DATA_BLOCK "Charge_1"	// DB 160
VERSION : 0.1
  STRUCT
   Recipe : INT ;
   batches : DINT ;
   Start : INT ;
   batchtime : DATE_AND_TIME ;
   header : ARRAY  [1 .. 7 ] OF INT ;
   BR : ARRAY  [1 .. 25 ] OF UDT 3;
  END_STRUCT ;	
BEGIN
   Recipe := 99;
   batches := L#8;
   Start := 2;
   BR[1].comp_nr := 4;
   BR[1].rated_val := 1.000000e+01;
   BR[1].real_val := 1.000681e+01;
   BR[3].comp_nr := 5;
   BR[3].rated_val := 5.000000e+00;
   BR[3].real_val := 4.986557e+00;
END_DATA_BLOCK

DATA_BLOCK "Charge_2"	// DB 161
VERSION : 0.1
  STRUCT
   Recipe : INT ;
   batches : DINT ;
   Start : INT ;
   batchtime : DATE_AND_TIME ;
   header : ARRAY  [1 .. 7 ] OF INT ;
   BR : ARRAY  [1 .. 25 ] OF UDT 3;
  END_STRUCT ;	
BEGIN
   Recipe := 199;
   batches := L#5;
   Start := 1;
   BR[1].comp_nr := 2;
   BR[1].rated_val := 2.000000e+00;
   BR[1].real_val := 3.009904e+00;
   BR[2].comp_nr := 3;
   BR[2].rated_val := 2.000000e+00;
   BR[2].real_val := 2.706667e+00;
   BR[3].comp_nr := 4;
   BR[3].rated_val := 2.000000e+00;
   BR[3].real_val := 1.864344e+00;
   BR[4].comp_nr := 6;
   BR[4].rated_val := 2.000000e-01;
   BR[4].real_val := 3.235633e-01;
   BR[5].comp_nr := 7;
   BR[5].rated_val := 2.000000e-01;
   BR[5].real_val := 4.058950e-01;
   BR[6].comp_nr := 8;
   BR[6].rated_val := 2.000000e-01;
   BR[6].real_val := 3.326198e-01;
   BR[7].comp_nr := 9;
   BR[7].rated_val := 2.000000e-01;
   BR[7].real_val := 3.507328e-01;
   BR[8].comp_nr := 10;
   BR[8].rated_val := 2.000000e-01;
   BR[8].real_val := 2.206488e-01;
   BR[9].comp_nr := 11;
   BR[9].rated_val := 2.000000e-01;
   BR[9].real_val := 2.684011e-01;
   BR[11].comp_nr := 5;
   BR[11].rated_val := 5.000000e+00;
   BR[11].real_val := 4.997788e+00;
END_DATA_BLOCK

DATA_BLOCK "Charge_3"	// DB 162
VERSION : 0.1
  STRUCT
   Recipe : INT ;
   batches : DINT ;
   Start : INT ;
   batchtime : DATE_AND_TIME ;
   header : ARRAY  [1 .. 7 ] OF INT ;
   BR : ARRAY  [1 .. 25 ] OF UDT 3;
  END_STRUCT ;	
BEGIN
   Recipe := 199;
   batches := L#6;
   Start := 1;
   BR[1].comp_nr := 2;
   BR[1].rated_val := 2.000000e+00;
   BR[1].real_val := 2.571896e+00;
   BR[2].comp_nr := 3;
   BR[2].rated_val := 2.000000e+00;
   BR[2].real_val := 2.482048e+00;
   BR[3].comp_nr := 4;
   BR[3].rated_val := 2.000000e+00;
   BR[3].real_val := 2.077733e+00;
   BR[4].comp_nr := 6;
   BR[4].rated_val := 2.000000e-01;
   BR[4].real_val := 3.013338e-01;
   BR[5].comp_nr := 7;
   BR[5].rated_val := 2.000000e-01;
   BR[5].real_val := 2.000659e-01;
   BR[6].comp_nr := 8;
   BR[6].rated_val := 2.000000e-01;
   BR[6].real_val := 2.165322e-01;
   BR[7].comp_nr := 9;
   BR[7].rated_val := 2.000000e-01;
   BR[7].real_val := 2.247653e-01;
   BR[8].comp_nr := 10;
   BR[8].rated_val := 2.000000e-01;
   BR[8].real_val := 2.247654e-01;
   BR[9].comp_nr := 11;
   BR[9].rated_val := 2.000000e-01;
   BR[9].real_val := 2.321752e-01;
   BR[11].comp_nr := 5;
   BR[11].rated_val := 5.000000e+00;
   BR[11].real_val := 5.065175e+00;
END_DATA_BLOCK

DATA_BLOCK "Charge_4"	// DB 163
VERSION : 0.1
  STRUCT
   Recipe : INT ;
   batches : DINT ;
   Start : INT ;
   batchtime : DATE_AND_TIME ;
   header : ARRAY  [1 .. 7 ] OF INT ;
   BR : ARRAY  [1 .. 25 ] OF UDT 3;
  END_STRUCT ;	
BEGIN
   Recipe := 199;
   batches := L#7;
   Start := 1;
   BR[1].comp_nr := 2;
   BR[1].rated_val := 2.000000e+00;
   BR[1].real_val := 1.841882e+00;
   BR[2].comp_nr := 3;
   BR[2].rated_val := 2.000000e+00;
   BR[2].real_val := 2.257428e+00;
   BR[3].comp_nr := 4;
   BR[3].rated_val := 2.000000e+00;
   BR[3].real_val := 1.942961e+00;
   BR[4].comp_nr := 6;
   BR[4].rated_val := 2.000000e-01;
   BR[4].real_val := 1.992425e-01;
   BR[5].comp_nr := 7;
   BR[5].rated_val := 2.000000e-01;
   BR[5].real_val := 1.728964e-01;
   BR[6].comp_nr := 8;
   BR[6].rated_val := 2.000000e-01;
   BR[6].real_val := 1.992425e-01;
   BR[7].comp_nr := 9;
   BR[7].rated_val := 2.000000e-01;
   BR[7].real_val := 2.124156e-01;
   BR[8].comp_nr := 10;
   BR[8].rated_val := 2.000000e-01;
   BR[8].real_val := 2.198255e-01;
   BR[9].comp_nr := 11;
   BR[9].rated_val := 2.000000e-01;
   BR[9].real_val := 2.082990e-01;
   BR[11].comp_nr := 5;
   BR[11].rated_val := 5.000000e+00;
   BR[11].real_val := 5.031482e+00;
END_DATA_BLOCK

DATA_BLOCK "Charge_5"	// DB 164
VERSION : 0.1
  STRUCT
   Recipe : INT ;
   batches : DINT ;
   Start : INT ;
   batchtime : DATE_AND_TIME ;
   header : ARRAY  [1 .. 7 ] OF INT ;
   BR : ARRAY  [1 .. 25 ] OF UDT 3;
  END_STRUCT ;	
BEGIN
   Recipe := 199;
   batches := L#1;
   Start := 2;
   BR[1].comp_nr := 2;
   BR[1].rated_val := 2.000000e+00;
   BR[1].real_val := 2.380969e+00;
   BR[2].comp_nr := 4;
   BR[2].rated_val := 2.000000e+00;
   BR[2].real_val := 2.066501e+00;
   BR[3].comp_nr := 6;
   BR[3].rated_val := 2.000000e-01;
   BR[3].real_val := 2.017125e-01;
   BR[4].comp_nr := 7;
   BR[4].rated_val := 2.000000e-01;
   BR[4].real_val := 1.901861e-01;
   BR[5].comp_nr := 8;
   BR[5].rated_val := 2.000000e-01;
   BR[5].real_val := 2.074757e-01;
   BR[6].comp_nr := 9;
   BR[6].rated_val := 2.000000e-01;
   BR[6].real_val := 2.140622e-01;
   BR[7].comp_nr := 10;
   BR[7].rated_val := 2.000000e-01;
   BR[7].real_val := 2.124156e-01;
   BR[8].comp_nr := 11;
   BR[8].rated_val := 2.000000e-01;
   BR[8].real_val := 2.025358e-01;
   BR[10].comp_nr := 5;
   BR[10].rated_val := 5.000000e+00;
   BR[10].real_val := 5.020251e+00;
END_DATA_BLOCK

DATA_BLOCK "Charge_6"	// DB 165
VERSION : 0.1
  STRUCT
   Recipe : INT ;
   batches : DINT ;
   Start : INT ;
   batchtime : DATE_AND_TIME ;
   header : ARRAY  [1 .. 7 ] OF INT ;
   BR : ARRAY  [1 .. 25 ] OF UDT 3;
  END_STRUCT ;	
BEGIN
   Recipe := 199;
   batches := L#2;
   Start := 2;
   BR[1].comp_nr := 2;
   BR[1].rated_val := 2.000000e+00;
   BR[1].real_val := 2.223735e+00;
   BR[2].comp_nr := 4;
   BR[2].rated_val := 2.000000e+00;
   BR[2].real_val := 2.066501e+00;
   BR[3].comp_nr := 6;
   BR[3].rated_val := 2.000000e-01;
   BR[3].real_val := 2.041824e-01;
   BR[4].comp_nr := 7;
   BR[4].rated_val := 2.000000e-01;
   BR[4].real_val := 2.848674e-01;
   BR[5].comp_nr := 8;
   BR[5].rated_val := 2.000000e-01;
   BR[5].real_val := 2.033591e-01;
   BR[6].comp_nr := 9;
   BR[6].rated_val := 2.000000e-01;
   BR[6].real_val := 2.041825e-01;
   BR[7].comp_nr := 10;
   BR[7].rated_val := 2.000000e-01;
   BR[7].real_val := 2.074757e-01;
   BR[8].comp_nr := 11;
   BR[8].rated_val := 2.000000e-01;
   BR[8].real_val := 2.017125e-01;
   BR[10].comp_nr := 5;
   BR[10].rated_val := 5.000000e+00;
   BR[10].real_val := 4.930403e+00;
END_DATA_BLOCK

DATA_BLOCK "Charge_7"	// DB 166
VERSION : 0.1
  STRUCT
   Recipe : INT ;
   batches : DINT ;
   Start : INT ;
   batchtime : DATE_AND_TIME ;
   header : ARRAY  [1 .. 7 ] OF INT ;
   BR : ARRAY  [1 .. 25 ] OF UDT 3;
  END_STRUCT ;	
BEGIN
   Recipe := 199;
   batches := L#3;
   Start := 2;
   BR[1].comp_nr := 2;
   BR[1].rated_val := 2.000000e+00;
   BR[1].real_val := 2.111425e+00;
   BR[2].comp_nr := 4;
   BR[2].rated_val := 2.000000e+00;
   BR[2].real_val := 1.886806e+00;
   BR[3].comp_nr := 6;
   BR[3].rated_val := 2.000000e-01;
   BR[3].real_val := 1.992425e-01;
   BR[4].comp_nr := 7;
   BR[4].rated_val := 2.000000e-01;
   BR[4].real_val := 2.404084e-01;
   BR[5].comp_nr := 8;
   BR[5].rated_val := 2.000000e-01;
   BR[5].real_val := 2.066524e-01;
   BR[6].comp_nr := 9;
   BR[6].rated_val := 2.000000e-01;
   BR[6].real_val := 2.017125e-01;
   BR[7].comp_nr := 10;
   BR[7].rated_val := 2.000000e-01;
   BR[7].real_val := 2.074757e-01;
   BR[8].comp_nr := 11;
   BR[8].rated_val := 2.000000e-01;
   BR[8].real_val := 1.992426e-01;
   BR[10].comp_nr := 5;
   BR[10].rated_val := 5.000000e+00;
   BR[10].real_val := 4.975327e+00;
END_DATA_BLOCK

DATA_BLOCK "Charge_8"	// DB 167
VERSION : 0.1
  STRUCT
   Recipe : INT ;
   batches : DINT ;
   Start : INT ;
   batchtime : DATE_AND_TIME ;
   header : ARRAY  [1 .. 7 ] OF INT ;
   BR : ARRAY  [1 .. 25 ] OF UDT 3;
  END_STRUCT ;	
BEGIN
   Recipe := 2;
   batches := L#11;
   Start := 1;
   BR[1].comp_nr := 3;
   BR[1].rated_val := 2.000000e+01;
   BR[1].real_val := -3.369296e-02;
END_DATA_BLOCK

DATA_BLOCK "Charge_9"	// DB 168
VERSION : 0.1
  STRUCT
   Recipe : INT ;
   batches : DINT ;
   Start : INT ;
   batchtime : DATE_AND_TIME ;
   header : ARRAY  [1 .. 7 ] OF INT ;
   BR : ARRAY  [1 .. 25 ] OF UDT 3;
  END_STRUCT ;	
BEGIN
   Recipe := 2;
   batches := L#12;
   Start := 1;
   BR[1].comp_nr := 6;
   BR[1].rated_val := 1.000000e+00;
END_DATA_BLOCK

DATA_BLOCK "Charge_10"	// DB 169
VERSION : 0.1
  STRUCT
   Recipe : INT ;
   batches : DINT ;
   Start : INT ;
   batchtime : DATE_AND_TIME ;
   header : ARRAY  [1 .. 7 ] OF INT ;
   BR : ARRAY  [1 .. 25 ] OF UDT 3;
  END_STRUCT ;	
BEGIN
   Recipe := 99;
   batches := L#7;
   Start := 2;
   BR[1].comp_nr := 4;
   BR[1].rated_val := 1.000000e+01;
   BR[1].real_val := 1.002927e+01;
   BR[3].comp_nr := 5;
   BR[3].rated_val := 5.000000e+00;
   BR[3].real_val := 4.952865e+00;
END_DATA_BLOCK

DATA_BLOCK "Recipes1-50"	// DB 333
TITLE = Data block for recipes 1-50
//it must be unlinked
//
AUTHOR : Fromm
VERSION : 1.0
  STRUCT
   Rezept : ARRAY  [1 .. 50 ] OF STRUCT
    step : ARRAY  [1 .. 25 ] OF UDT 1;
   END_STRUCT ;
  END_STRUCT ;	
BEGIN
END_DATA_BLOCK

DATA_BLOCK "Recipes51-100"	// DB 334
TITLE = Data block for recipes 51-100
//it must be unlinked
//
VERSION : 0.0
  STRUCT
   Rezept : ARRAY  [51 .. 100 ] OF STRUCT
    step : ARRAY  [1 .. 25 ] OF UDT 1;
   END_STRUCT ;
  END_STRUCT ;	
BEGIN
END_DATA_BLOCK

DATA_BLOCK "Recipes101-150"	// DB 335
TITLE = Data block for recipes 101-150
//it must be unlinked
//
AUTHOR : Fromm
VERSION : 1.0
  STRUCT
   Rezept : ARRAY  [101 .. 150 ] OF STRUCT
    step : ARRAY  [1 .. 25 ] OF UDT 1;
   END_STRUCT ;
  END_STRUCT ;	
BEGIN
END_DATA_BLOCK

DATA_BLOCK "Recipes151-200"	// DB 336
TITLE = Data block for recipes 151-200
//it must be unlinked
//
AUTHOR : Fromm
VERSION : 1.0
  STRUCT
   Rezept : ARRAY  [151 .. 200 ] OF STRUCT
    step : ARRAY  [1 .. 25 ] OF UDT 1;
   END_STRUCT ;
  END_STRUCT ;	
BEGIN
END_DATA_BLOCK

ORGANIZATION_BLOCK OB 1
TITLE = "Main Program Sweep (Cycle)"
VERSION : 0.1
VAR_TEMP
  OB1_EV_CLASS : BYTE ;	//Bits 0-3 = 1 (Coming event), Bits 4-7 = 1 (Event class 1)
  OB1_SCAN_1 : BYTE ;	//1 (Cold restart scan 1 of OB 1), 3 (Scan 2-n of OB 1)
  OB1_PRIORITY : BYTE ;	//Priority of OB Execution
  OB1_OB_NUMBR : BYTE ;	//1 (Organization block 1, OB1)
  OB1_RESERVED_1 : BYTE ;	//Reserved for system
  OB1_RESERVED_2 : BYTE ;	//Reserved for system
  OB1_PREV_CYCLE : INT ;	//Cycle time of previous OB1 scan (milliseconds)
  OB1_MIN_CYCLE : INT ;	//Minimum cycle time of OB1 (milliseconds)
  OB1_MAX_CYCLE : INT ;	//Maximum cycle time of OB1 (milliseconds)
  OB1_DATE_TIME : DATE_AND_TIME ;	//Date and time OB1 started
END_VAR
BEGIN
NETWORK
TITLE =
      A     "permanent_0";
      R     "permanent_0";
      AN    "permanent_1";
      S     "permanent_1";
      A     "Restart_Timer";
      =     "StartupTimer";
      A     "permanent_1";
      FP    M 200.0;
      =     "CPU_Restart";
NETWORK
TITLE =
      CALL  "errors_horn";
      CALL  "start_lamps";
      CALL  "dos_comp_1";
      CALL  "dos_comp_2";
      CALL  "dos_comp_5";
      CALL  "dos_comp_6_SS";
      CALL  "dos_comp_7";
      CALL  "dos_comp_8";
      CALL  "dos_comp_9";
      CALL  "dos_comp_10";
      CALL  "dos_comp_11";
      CALL  "dos_comp_12";
      CALL  "discharge_main_scale";
      CALL  "discharge_sub_scale";
      CALL  "agit_MS";
      CALL  "aigt_level_storage1";
      CALL  "aigt_level_storage2";
      CALL  "filling_vat";
      CALL  "filling_coater";
      CALL  "coater circ";
      CALL  "control_FC";
      CALL  "Hand_OP_FC";
END_ORGANIZATION_BLOCK

ORGANIZATION_BLOCK "I/O_FLT1"	// OB 82
TITLE = "I/O Point Fault"
VERSION : 0.1
VAR_TEMP
  OB82_EV_CLASS : BYTE ;	//16#39, Event class 3, Entering event state, Internal fault event
  OB82_FLT_ID : BYTE ;	//16#XX, Fault identifcation code
  OB82_PRIORITY : BYTE ;	//Priority of OB Execution
  OB82_OB_NUMBR : BYTE ;	//82 (Organization block 82, OB82)
  OB82_RESERVED_1 : BYTE ;	//Reserved for system
  OB82_IO_FLAG : BYTE ;	//Input (01010100), Output (01010101)
  OB82_MDL_ADDR : WORD ;	//Base address of module with fault
  OB82_MDL_DEFECT : BOOL ;	//Module defective
  OB82_INT_FAULT : BOOL ;	//Internal fault
  OB82_EXT_FAULT : BOOL ;	//External fault
  OB82_PNT_INFO : BOOL ;	//Point information
  OB82_EXT_VOLTAGE : BOOL ;	//External voltage low
  OB82_FLD_CONNCTR : BOOL ;	//Field wiring connector missing
  OB82_NO_CONFIG : BOOL ;	//Module has no configuration data
  OB82_CONFIG_ERR : BOOL ;	//Module has configuration error
  OB82_MDL_TYPE : BYTE ;	//Type of module
  OB82_SUB_MDL_ERR : BOOL ;	//Sub-Module is missing or has error
  OB82_COMM_FAULT : BOOL ;	//Communication fault
  OB82_MDL_STOP : BOOL ;	//Module is stopped
  OB82_WTCH_DOG_FLT : BOOL ;	//Watch dog timer stopped module
  OB82_INT_PS_FLT : BOOL ;	//Internal power supply fault
  OB82_PRIM_BATT_FLT : BOOL ;	//Primary battery is in fault
  OB82_BCKUP_BATT_FLT : BOOL ;	//Backup battery is in fault
  OB82_RESERVED_2 : BOOL ;	//Reserved for system
  OB82_RACK_FLT : BOOL ;	//Rack fault, only for bus interface module
  OB82_PROC_FLT : BOOL ;	//Processor fault
  OB82_EPROM_FLT : BOOL ;	//EPROM fault
  OB82_RAM_FLT : BOOL ;	//RAM fault
  OB82_ADU_FLT : BOOL ;	//ADU fault
  OB82_FUSE_FLT : BOOL ;	//Fuse fault
  OB82_HW_INTR_FLT : BOOL ;	//Hardware interupt input in fault
  OB82_RESERVED_3 : BOOL ;	//Reserved for system
  OB82_DATE_TIME : DATE_AND_TIME ;	//Date and time OB82 started
END_VAR
BEGIN
// (block stored without names or comments; labels and parameter names are numbered)
END_ORGANIZATION_BLOCK

ORGANIZATION_BLOCK "RACK_FLT"	// OB 86
TITLE = "Loss Of Rack Fault"
VERSION : 0.1
VAR_TEMP
  OB86_EV_CLASS : BYTE ;	//16#38/39 Event class 3
  OB86_FLT_ID : BYTE ;	//16#C1/C4/C5, Fault identifcation code
  OB86_PRIORITY : BYTE ;	//Priority of OB Execution
  OB86_OB_NUMBR : BYTE ;	//86 (Organization block 86, OB86)
  OB86_RESERVED_1 : BYTE ;	//Reserved for system
  OB86_RESERVED_2 : BYTE ;	//Reserved for system
  OB86_MDL_ADDR : WORD ;	//Base address of IM module in rack with fault
  OB86_RACKS_FLTD : ARRAY  [0 .. 31 ] OF BOOL ;	//Racks in fault
  OB86_DATE_TIME : DATE_AND_TIME ;	//Date and time OB86 started
END_VAR
BEGIN
// (block stored without names or comments; labels and parameter names are numbered)
END_ORGANIZATION_BLOCK

ORGANIZATION_BLOCK "COMPLETE RESTART"	// OB 100
TITLE = "Complete Restart"
VERSION : 0.1
VAR_TEMP
  OB100_EV_CLASS : BYTE ;	//16#13, Event class 1, Entering event state, Event logged in diagnostic buffer
  OB100_STRTUP : BYTE ;	//16#81/82/83/84 Method of startup
  OB100_PRIORITY : BYTE ;	//27 (Priority of 1 is lowest)
  OB100_OB_NUMBR : BYTE ;	//100 (Organization block 100, OB100)
  OB100_RESERVED_1 : BYTE ;	//Reserved for system
  OB100_RESERVED_2 : BYTE ;	//Reserved for system
  OB100_STOP : WORD ;	//Event that caused CPU to stop (16#4xxx)
  OB100_STRT_INFO : DWORD ;	//Information on how system started
  OB100_DATE_TIME : DATE_AND_TIME ;	//Date and time OB100 started
END_VAR
BEGIN
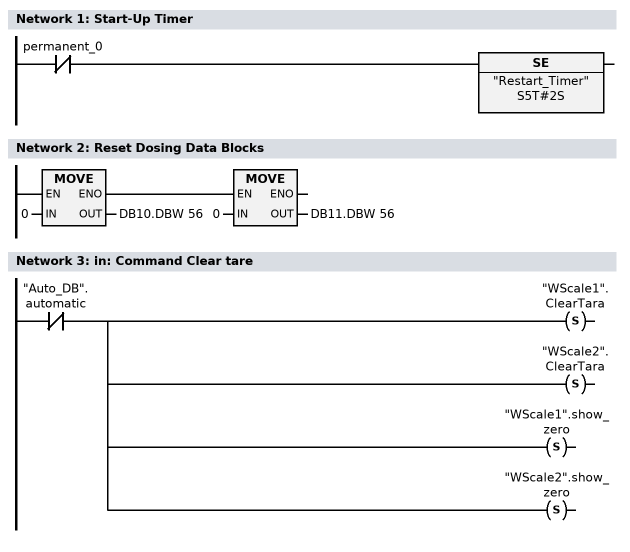
NETWORK
TITLE = Start-Up Timer
      AN    "permanent_0";
      L     S5T#2S;
      SE    "Restart_Timer";
NETWORK
TITLE = Reset Dosing Data Blocks
      A(;
      L     0;
      T     DB10.DBW 56;
      SET;
      SAVE;
      CLR;
      A     BR;
      );
      JNB   _001;
      L     0;
      T     DB11.DBW 56;
_001: NOP   0;
NETWORK
TITLE = in: Command Clear tare
      AN    "Auto_DB".automatic;
      S     "WScale1".ClearTara;
      S     "WScale2".ClearTara;
      S     "WScale1".show_zero;
      S     "WScale2".show_zero;
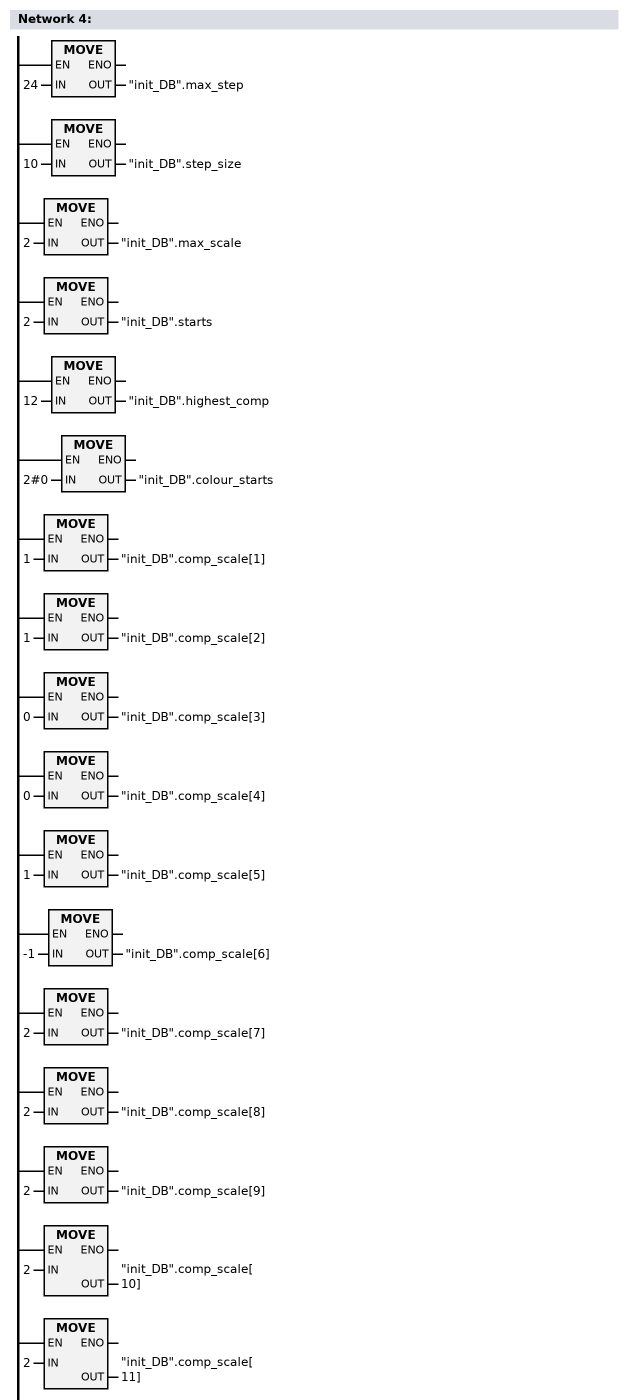
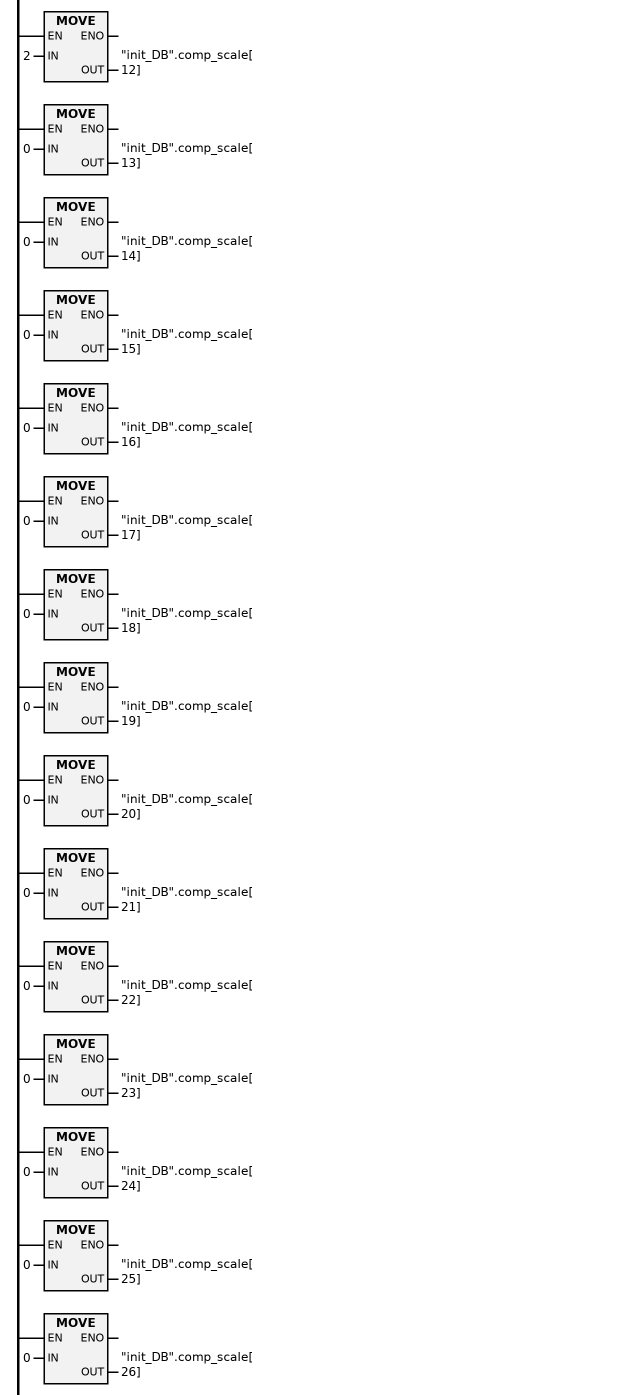
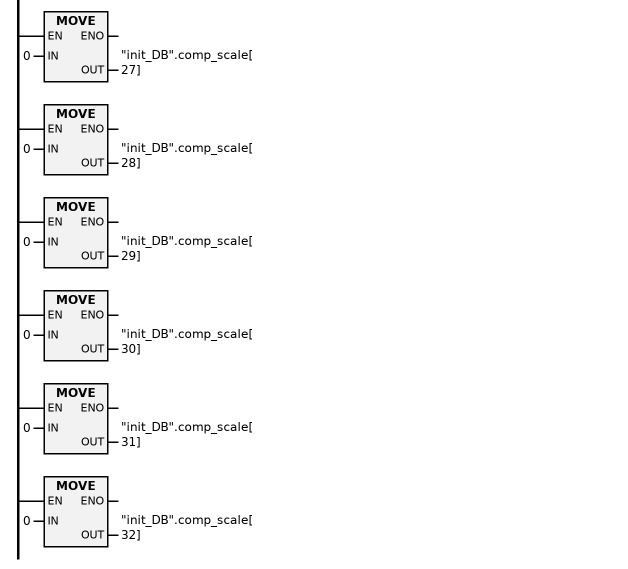
NETWORK
TITLE =
      L     24;
      T     "init_DB".max_step;
      L     10;
      T     "init_DB".step_size;
      L     2;
      T     "init_DB".max_scale;
      L     2;
      T     "init_DB".starts;
      L     12;
      T     "init_DB".highest_comp;
      L     2#0;
      T     "init_DB".colour_starts;
// 1: main scale
// 2: sub scale
// 3: color scale
      L     1;
      T     "init_DB".comp_scale[1];
      L     1;
      T     "init_DB".comp_scale[2];
      L     0;
      T     "init_DB".comp_scale[3];
      L     0;
      T     "init_DB".comp_scale[4];
      L     1;
      T     "init_DB".comp_scale[5];
      L     -1;
      T     "init_DB".comp_scale[6];
      L     2;
      T     "init_DB".comp_scale[7];
      L     2;
      T     "init_DB".comp_scale[8];
      L     2;
      T     "init_DB".comp_scale[9];
      L     2;
      T     "init_DB".comp_scale[10];
      L     2;
      T     "init_DB".comp_scale[11];
      L     2;
      T     "init_DB".comp_scale[12];
      L     0;
      T     "init_DB".comp_scale[13];
      L     0;
      T     "init_DB".comp_scale[14];
      L     0;
      T     "init_DB".comp_scale[15];
      L     0;
      T     "init_DB".comp_scale[16];
      L     0;
      T     "init_DB".comp_scale[17];
      L     0;
      T     "init_DB".comp_scale[18];
      L     0;
      T     "init_DB".comp_scale[19];
      L     0;
      T     "init_DB".comp_scale[20];
      L     0;
      T     "init_DB".comp_scale[21];
      L     0;
      T     "init_DB".comp_scale[22];
      L     0;
      T     "init_DB".comp_scale[23];
      L     0;
      T     "init_DB".comp_scale[24];
      L     0;
      T     "init_DB".comp_scale[25];
      L     0;
      T     "init_DB".comp_scale[26];
      L     0;
      T     "init_DB".comp_scale[27];
      L     0;
      T     "init_DB".comp_scale[28];
      L     0;
      T     "init_DB".comp_scale[29];
      L     0;
      T     "init_DB".comp_scale[30];
      L     0;
      T     "init_DB".comp_scale[31];
      L     0;
      T     "init_DB".comp_scale[32];
NETWORK
TITLE = init CP Gravimet
      L     160;
      T     "init_DB".CP_DB_MIN;
      L     10;
      T     "init_DB".CP_DB_ANZ;
      L     "HMI_DB".CP_DB_WRITE;
      L     "init_DB".CP_DB_MIN;
      <I;
      JC    err1;
      L     "init_DB".CP_DB_MIN;
      L     "init_DB".CP_DB_ANZ;
      +I;
      L     "HMI_DB".CP_DB_WRITE;
      TAK;
      >=I;
      JC    err1;
      JU    go1;
err1: L     "init_DB".CP_DB_MIN;
      T     "HMI_DB".CP_DB_WRITE;
go1:  NOP   0;
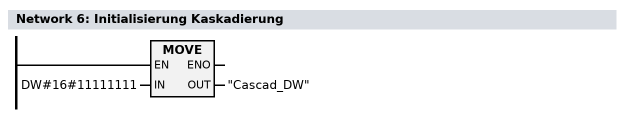
NETWORK
TITLE = Initialisierung Kaskadierung
      L     DW#16#11111111;
      T     "Cascad_DW";
END_ORGANIZATION_BLOCK

ORGANIZATION_BLOCK "PROG_ERR"	// OB 121
TITLE = "Programming Error"
VERSION : 0.1
VAR_TEMP
  OB121_EV_CLASS : BYTE ;	//16#25, Event class 2, Entering event state, Internal fault event
  OB121_SW_FLT : BYTE ;	//16#XX Software programming fault
  OB121_PRIORITY : BYTE ;	//Priority of OB Execution
  OB121_OB_NUMBR : BYTE ;	//121 (Organization block 121, OB121)
  OB121_BLK_TYPE : BYTE ;	//16#88/8A/8B/8C/8E Type of block fault occured in
  OB121_RESERVED_1 : BYTE ;	//Reserved for system
  OB121_FLT_REG : WORD ;	//16#XX Specific register that caused fault
  OB121_BLK_NUM : WORD ;	//Number of block that programming fault occured in
  OB121_PRG_ADDR : WORD ;	//Address in block where programming fault occured
  OB121_DATE_TIME : DATE_AND_TIME ;	//Date and time OB121 started
END_VAR
BEGIN
// (block stored without names or comments; labels and parameter names are numbered)
END_ORGANIZATION_BLOCK

ORGANIZATION_BLOCK "MOD_ERR"	// OB 122
TITLE = "Module Access Error"
VERSION : 0.1
VAR_TEMP
  OB122_EV_CLASS : BYTE ;	//16#29, Event class 2, Entering event state, Internal fault event
  OB122_SW_FLT : BYTE ;	//16#XX Software error code
  OB122_PRIORITY : BYTE ;	//Priority of OB Execution
  OB122_OB_NUMBR : BYTE ;	//122 (Organization block 122, OB122)
  OB122_BLK_TYPE : BYTE ;	//16#88/8C/8E Type of block fault occured in
  OB122_MEM_AREA : BYTE ;	//Memory area where access error occured
  OB122_MEM_ADDR : WORD ;	//Memory address where access error occured
  OB122_BLK_NUM : WORD ;	//Block number in which error occured
  OB122_PRG_ADDR : WORD ;	//Program address where error occured
  OB122_DATE_TIME : DATE_AND_TIME ;	//Date and time OB1 started
END_VAR
BEGIN
// (block stored without names or comments; labels and parameter names are numbered)
END_ORGANIZATION_BLOCK

FUNCTION_BLOCK FB 2
//know_how_protect
//
VERSION : 0.1
VAR_INPUT
  scale_nr : INT ;
  Work_DB : INT ;
  Weigh_DB : INT ;
  mix_timer : TIMER ;
END_VAR
VAR_IN_OUT
  step_scale1 : INT ;
  step_scale2 : INT ;
  step_scale3 : INT ;
  step_scale4 : INT ;
  Dosi_Bits : DINT ;
END_VAR
VAR
  DB_ptr : INT ;
  rated_val : REAL ;
  dosi_val_fine : REAL ;
  dosi_val_coarse : REAL ;
  enable : BOOL ;
  inc_step : BOOL ;
  dosing : BOOL ;
  dosi_coarse : BOOL ;
  dosi_fine : BOOL ;
  cancel : BOOL ;
  discharge : BOOL ;	//out: discharge scale
  wait_still : BOOL ;
  dosi_err : BOOL ;
  dosi_time_err : BOOL ;
  quit_wait : BOOL ;
  redosi : BOOL ;
  mix_time : BOOL ;
  stop : BOOL ;
  clean_out : BOOL ;
  ScaleDosi_Bit : DINT ;
  OwnStep : INT ;
  Status : INT ;
  Rated_Sum : REAL ;
  comp_nr : INT ;
END_VAR
VAR_TEMP
  comp_ok : BOOL ;
  Standstill : BOOL ;
  empty : BOOL ;
  time_empty : BOOL ;
  DosiControl : BOOL ;
  TareScale : BOOL ;
  StepTime : BOOL ;
  ClearTara : BOOL ;
  Temp : INT ;
  NetWeight : REAL ;
  StepPtr : DINT ;
  ScalePtr1 : DINT ;
  scalePtr2 : DINT ;
  scalePtr3 : DINT ;
  scalePtr4 : DINT ;
  t_comp_nr : INT ;
  t_scale : INT ;
  t_spuel : BOOL ;
  start_nr : BYTE ;
END_VAR
BEGIN
NETWORK
TITLE = Read Weighing datas
      L     0;
      T     LB 0;
      AN    #enable;
      BEC;
      L     #Weigh_DB;
      T     #Temp;
      OPN   DB [#Temp];
      L     DBD 88;
      T     #NetWeight;
      A     DBX 58.0;
      =     #Standstill;
      A     DBX 58.3;
      =     #empty;
      A     DBX 58.4;
      =     #time_empty;
      AN    #quit_wait;
      R     #dosi_time_err;
      A     DBX 58.5;
      =     #DosiControl;
      L     0;
      T     #Status;
      A     DBX 58.6;
      =     #StepTime;
      JCN   nost;
      L     10;
      T     #Status;
nost: NOP   0;
      L     #ScaleDosi_Bit;
      L     #Dosi_Bits;
      OD;
      T     #Dosi_Bits;
      A     #cancel;
      R     #quit_wait;
      S     #ClearTara;
NETWORK
TITLE = Jump
      A     #cancel;
      AN    #dosing;
      JC    tend;
      A     #wait_still;
      JC    stil;
      A     #quit_wait;
      JC    end;
      A     #dosi_err;
      JC    t_ok;
      A     #dosing;
      JC    dosi;
      A     #mix_time;
      JC    time;
NETWORK
TITLE = increment own step
      L     #scale_nr;
      L     P#2.0;
      *D;
      L     P#6.0;
      +D;
      T     #StepPtr;
      AN    #inc_step;
      JC    ninc;
      R     #inc_step;
      L     DB1.DBW 0;
      L     #OwnStep;
      ==I;
//      U     #empty
      JC    tend;
// Entleeren, wenn Waage zum Schluß nicht leer (Entleeren vergessen)
// noch nicht ausgereift (Synchronisation fehlt)
//      L     "init_DB".max_step
//      L     #OwnStep
//      ==I   
//      UN    #empty
//      SPB   disc
      INC   1;
      T     DIW [#StepPtr];
      T     #OwnStep;
ninc: NOP   0;
NETWORK
TITLE = calculate pointer
//Vorerst nicht verwendet
      L     #OwnStep;
      DEC   1;
      L     DB1.DBW 2;
      *D;
      SLD   3;
      LAR1;
      L     0;
      L     #step_scale1;
      ==I;
      JC    z1;
      DEC   1;
      L     DB1.DBW 2;
      *D;
      SLD   3;
z1:   T     #ScalePtr1;
      L     0;
      L     #step_scale2;
      ==I;
      JC    z2;
      DEC   1;
      L     DB1.DBW 2;
      *D;
      SLD   3;
z2:   T     #scalePtr2;
      L     0;
      L     #step_scale3;
      ==I;
      JC    z3;
      DEC   1;
      L     DB1.DBW 2;
      *D;
      SLD   3;
z3:   T     #scalePtr3;
      L     0;
      L     #step_scale4;
      ==I;
      JC    z4;
      DEC   1;
      L     DB1.DBW 2;
      *D;
      SLD   3;
z4:   T     #scalePtr4;
NETWORK
TITLE = Sync all other scales
      L     #Work_DB;
      T     #Temp;
      OPN   DB [#Temp];
      L     DBW [AR1,P#2.0];	// comp no.
      T     #t_comp_nr;
      CALL  FC 85 (
           component                := #t_comp_nr,
           scale_nr                 := #t_scale);	//WAAGE FUER KOMPONENTE ABFRAGEN
      A(;
      L     W#16#FF;
      L     #t_scale;
      ==I;	// Spülkomponente
      );
      A(;
      L     #scale_nr;
      L     2;	// Subwaage
      ==I;
      );
      =     #t_spuel;
      A(;
      L     #step_scale1;
      L     #OwnStep;
      <=I;
      );
      A     #t_spuel;
      JC    end;
      L     DBW [AR1,P#0.0];	// Action
      SRW   8;
      L     #scale_nr;
      <>I;
      S     #inc_step;	// nicht für diese Waage
      JC    end;
//      SPA   sync                        // kein Paralleldosieren der waagen
      L     16;
      T     #Status;
      A(;
      L     DBW [AR1,P#0.0];	// Action
      L     W#16#FF;
      AW;
      L     1;	// dosieren
      <=I;
      );
      A(;
      L     #scale_nr;
      L     2;	// nur Subwaage darf parallel
      ==I;
      );
      JC    tar;	// Dosieren ohne Synchronisation (parallel)
      A(;
      L     #step_scale1;
      L     #OwnStep;
      >=I;
      );
      A(;
      L     #step_scale2;
      L     #OwnStep;
      >=I;
      );
      A(;
      L     #step_scale3;
      L     #OwnStep;
      >=I;
      );
      A(;
      L     #step_scale4;
      L     #OwnStep;
      >=I;
      );
      JCN   end;
      NOP   0;
NETWORK
TITLE = step for this scale?
      L     #Work_DB;
      T     #Temp;
      OPN   DB [#Temp];
      L     DBW [AR1,P#0.0];	// Action
      L     W#16#FF;	// nur das untere Byte
      AW;
      T     #Temp;
      L     1;	// dosieren
      <=I;
      JC    tar;
      L     #Temp;	// Action
      L     2;
      ==I;	// mixing?
      JC    mix;
      L     #Temp;	// Action
      L     3;
      ==I;	// discharge?
      JC    disc;
      L     #Temp;	// Action
      L     4;
      ==I;	// discharge cleaning
      S     #clean_out;
      JC    disc;
      S     #inc_step;	// keine der Aktionen
      JU    end;
NETWORK
TITLE = Action: mixing
mix:  L     #OwnStep;
      DEC   1;
      L     DB1.DBW 2;
      *I;
      SLD   3;
      LAR1;
      L     #Work_DB;
      T     #Temp;
      OPN   DB [#Temp];
// Subwaage mit Entleeren
      L     DBW [AR1,P#0.0];	// Action
      L     W#16#FF;
      AW;
      L     0;	// 0 =mit entleeren
      <>I;
      JC    mix2;
      L     W#16#3;
      L     DBW [AR1,P#0.0];
      OW;
      T     DBW [AR1,P#0.0];
      JU    end;
mix2: NOP   0;
// Ende
      L     0;
      L     DBW [AR1,P#4.0];	// mixing time
      ==I;
      S     #inc_step;
      JC    end;
      S     #mix_time;
      JU    end;
time: L     12;
      T     #Status;
      T     LD 34;
      TAK;
      T     LD 38;
      L     #mix_timer;
      T     LW 42;
      L     LD 38;
      L     LD 34;
      AN    T [LW 42];
      BEC;
      SET;
      R     #mix_time;
      S     #inc_step;
      L     0;
      T     #rated_val;
      T     #comp_nr;
      JU    end;
NETWORK
TITLE = Action: discharge scale
disc: L     4;
      T     #Status;
      L     #Rated_Sum;
      T     #rated_val;
      S     #ClearTara;
      A     #empty;
      AN    #time_empty;
      JCN   not;
      L     15;
      T     #Status;
not:  AN    #time_empty;
      =     #discharge;
      JC    end;
      R     #clean_out;
      L     0;
      T     #Rated_Sum;
      JU    mix;
NETWORK
TITLE = tare scale
tar:  L     8;
      T     #Status;
      L     DBW [AR1,P#2.0];	// comp no.
      T     #comp_nr;
      L     DBD [AR1,P#6.0];
      T     #rated_val;
//      CALL  "comp_scale"
//       component:=#comp_nr
//       scale_nr :=#Temp
//      L     #Temp
//      L     #scale_nr
//      <>I   
//      S     #inc_step
//      SPB   end
      L     9;
      T     #Status;
      AN    #Standstill;
      JC    end;
      L     #rated_val;
      L     #Rated_Sum;
      +R;
      T     #Rated_Sum;
      L     #comp_nr;
      L     30;
      +I;
      T     #DB_ptr;
      T     #Temp;
      OPN   DB [#Temp];
      L     1;
      T     #ScaleDosi_Bit;
      L     #comp_nr;
      DEC   1;
      L     #ScaleDosi_Bit;
      SLD;
      T     #ScaleDosi_Bit;
      L     #Dosi_Bits;
      OD;
      T     #Dosi_Bits;
      L     #rated_val;
      L     DBD 16;	// Nachlauf
      -R;
      JP    f_ok;
      L     0.000000e+00;
      T     DBD 16;
      L     #rated_val;
f_ok: T     #dosi_val_fine;
      L     DBD 8;	// grob/fein
      -R;
      JP    c_ok;
//      L     DBD    0
//      T     DBD    8
      L     #dosi_val_fine;
c_ok: T     #dosi_val_coarse;
// DosiTime at CompDatas
      L     DBW 20;
      L     #Weigh_DB;
      T     #Temp;
      TAK;
      OPN   DB [#Temp];
      T     DBW 116;
// End  DosiTime at CompDatas 
      S     #TareScale;
      S     #dosing;
      JU    end;
NETWORK
TITLE = dosing
dosi: A     #cancel;
      JC    t_ok;
      AN    #dosi_fine;
      A     #StepTime;
      JC    end;
      O     #stop;
      O     #DosiControl;
      S     #quit_wait;
      R     #dosi_coarse;
      R     #dosi_fine;
      S     #dosi_time_err;
      JC    end;
      L     #NetWeight;
      L     #dosi_val_fine;
      <R;
      =     #dosi_fine;
      L     #NetWeight;
      L     #dosi_val_coarse;
      <R;
      =     #dosi_coarse;
      L     3;
      A     #dosi_fine;
      AN    #dosi_coarse;
      JC    tran;
      L     2;
tran: T     #Status;
      O     #dosi_coarse;
      O     #dosi_fine;
      JC    end;
NETWORK
TITLE = drip_flow
      A     #StepTime;
      JC    end;
stil: AN    #Standstill;
      =     #wait_still;
      JC    end;
      A     #redosi;
      JC    tol;
      L     #DB_ptr;
      T     #Temp;
      OPN   DB [#Temp];
      L     #NetWeight;
      L     #rated_val;
      -R;
      L     5.000000e-01;
      *R;
      L     DBD 16;
      +R;
      JP    npos;
      L     0.000000e+00;
npos: T     DBD 16;
NETWORK
TITLE = Tolerance
tol:  R     #redosi;
      L     #DB_ptr;
      T     #Temp;
      OPN   DB [#Temp];
      L     #NetWeight;
      L     #rated_val;
      -R;
      JP    tpos;
      S     #redosi;	// evtl nachdos
      ABS;
tpos: L     DBD 12;	// tolerance
      <R;	// Abweichung < Toleranz
      JC    t_ok;
      AN    #redosi;
      S     #dosi_err;
      S     #quit_wait;
      JC    end;
// Nachdosieren
      L     #rated_val;	//neu, Sollwert
      L     DBD 12;	//Toleranz
      -R;
      T     #dosi_val_fine;
      JU    end;
t_ok: R     #dosi_err;
NETWORK
TITLE = dosing end
      R     #dosing;
      CALL  FC 65 (
           start_nr                 := DB21.DBB 6,
           scale_nr                 := #scale_nr,
           step                     := #OwnStep,
           comp                     := #comp_nr,
           rated_val                := #rated_val,
           real_val                 := #NetWeight);
      L     #ScaleDosi_Bit;
      INVD;
      L     #Dosi_Bits;
      AD;
      T     #Dosi_Bits;
      L     0;
      T     #ScaleDosi_Bit;
      A     #cancel;
      JC    tend;
      JU    mix;
NETWORK
TITLE =
tend: L     0;
      T     DIW 34;
      T     #OwnStep;
      T     #Rated_Sum;
      T     #rated_val;
      T     #comp_nr;
NETWORK
TITLE =
end:  A     #mix_time;
      ITB;
      OW    W#16#2000;
      T     LD 34;
      TAK;
      T     LD 38;
      L     #mix_timer;
      T     LW 42;
      L     LD 38;
      L     LD 34;
      SD    T [LW 42];
NETWORK
TITLE = Write Weighing Datas
      L     #Weigh_DB;
      T     #Temp;
      OPN   DB [#Temp];
      A     #TareScale;
      S     DBX 57.0;
      A     #ClearTara;
      S     DBX 57.1;
      A     #dosi_fine;
      =     DBX 57.3;
      A     #discharge;
      =     DBX 57.4;
END_FUNCTION_BLOCK

FUNCTION_BLOCK FB 111
TITLE = Wiegebaustein mit Siwarex CS
//
//Version: 1.0 (Beta-Version)
//Entwicklung: 10.11.2010 Stefan Michel
//
//Bemerkungen: -Baustein für Funktionstests im Haus freigegeben
//             
//
//Änderungen:
//
//
AUTHOR : Michel
VERSION : 1.0
VAR_INPUT
  ADRESSE : INT ;	//Adresse der Siwarex Baugruppe (Hardwarekonfig)
  ABZUGSWAAGE : BOOL ;	//Zuwaage:0;          Abzugswaage:1
  KAS_SIWAREX : BOOL ;	//Kaskadierung Siwarex (wird nur angesprochen, wenn 1 (Zugriffe optimieren)
  CPU_Start_Bit : BOOL ;	//Ein Bit das beim CPU-Start für 1Zyklus den Zustand 1 hat
  ANLAUFTIMER : BOOL ;	//Anlauftimer der CPU
  Quitt : BOOL ;	//Quittiermerker
  StillTimer : TIMER ;	//Timer for Standstill
  EmptyTimer : TIMER ;	//Timer for emptyTime
  DosiControlTimer : TIMER ;	//Timer for dosiControl
  StepTimer : TIMER ;	//Timer for StepTime
END_VAR
VAR_IN_OUT
  SYNCHRON_ERR : BOOL ;	//Synchroner Fehler der SIWAREX
  ASYNCHRON_ERR : BOOL ;	//Asynchroner Fehler der SIWAREX
  SIWA_ERR : BOOL ;	//Siwarex liefert keine neuen Messwerte/oder Kommunikation gestört
  SFB_ERR : BOOL ;	//Fehler bei der SFB-Bearbeitung
  BUSY : BOOL ;	//BIN BESCHÄFTIGT!  Es wird gerade ein SFB abgearbeitet
END_VAR
VAR
  Reserve : ARRAY  [0 .. 1 ] OF //Reserve
  BYTE ;
  AdjustDatas : STRUCT 	//DataRecords 3 and 4
   Zero_set_val_NV : WORD ;	//nicht verwendet
   Meanval_filt_NV : BOOL ;	//nicht verwendet
   EEPROM_NV : BOOL ;	//nicht verwendet
   Chan_active_NV : BOOL ;	//nicht verwendet
   Free1_NV : BOOL ;	//nicht verwendet
   Free2_NV : BOOL ;	//nicht verwendet
   Free3_NV : BOOL ;	//nicht verwendet
   Free4_NV : BOOL ;	//nicht verwendet
   Free5_NV : BOOL ;	//nicht verwendet
   LoadCell1_NV : BOOL ;	//nicht verwendet
   LoadCell2_NV : BOOL ;	//nicht verwendet
   Comma1_NV : BOOL ;	//nicht verwendet
   Comma2_NV : BOOL ;	//nicht verwendet
   Comma3_NV : BOOL ;	//nicht verwendet
   Filter1_NV : BOOL ;	//nicht verwendet
   Filter2_NV : BOOL ;	//nicht verwendet
   Filter3_NV : BOOL ;	//nicht verwendet
   Digit0 : WORD ;	//Adjustment digits dead load
   Digit1 : WORD  := W#16#EA60;	//Adjustment digits Adjustment weight
   AdjustWeight : INT  := 2000;	//Adjustment weight
  END_STRUCT ;
  Reserve_1 : ARRAY  [0 .. 9 ] OF //Reserve
  BYTE ;
  Command : WORD ;	//DataRecords 11 and 12 Command (1 zero point;2 adjustment point; 3 set zero)
  Reserve_2 : ARRAY  [0 .. 7 ] OF //Reserve
  BYTE ;
  ActDatas : STRUCT 	//DataRecords 31 and 32
   Gross : INT ;	//Grossweight für Dosierzeitkontrolle und Stillstandskontrolle
   Status_NV : BYTE ;	//nicht verwendet
   MeasVal_NV : BYTE ;	//nicht verwendet
   Digits : WORD ;
   Asynch_Err_NV : WORD ;	//nicht verwendet
   Synch_Err_NV : WORD ;	//nicht verwendet
  END_STRUCT ;
  ReadAdjust : BOOL ;	//Bit Justagedaten lesen
  Res_1 : BOOL ;
  WriteAdjust : BOOL ;	//Bit Justagedaten schreiben
  Res_2 : BOOL ;
  WriteCommand : BOOL ;	//Write Siwarex command
  Res_3 : BOOL ;
  Res_4 : BOOL ;
  Res_5 : BOOL ;
  TareScale : BOOL ;	//Bit Waage tarieren
  ClearTara : BOOL ;	//Bit lösche Taraspeicher - Zeige Inhalt der Waage
  show_zero : BOOL ;	//zeige absoluten Inhalt der Waage an
  dosing : BOOL ;	//Waage ist in der Dosierung
  discharge : BOOL ;	//Waage ist in der Entleerung
  Res_6 : BOOL ;
  Res_7 : BOOL ;
  Res_8 : BOOL ;
  Standstill : BOOL ;	//Stillstand Waage
  Overload : BOOL ;	//Waage ist überlastet
  no_zero : BOOL ;	//Nullfehler (AbsGewicht > Nullwert)
  empty : BOOL ;	//Erkennung Waage leer --> Leerzeit startet
  time_empty : BOOL ;	//Waage leer und Leerzeit abgelaufen
  DosiControl : BOOL ;	//Dosierzeitfehler
  StepTime : BOOL ;	//Fortschaltezeit läuft
  DosiControl_OldVal : INT ;	//Dosierzeitkontrolle alter Wert
  StandStill_OldVal : INT ;	//Stillstandskontrolle alter Wert
  SiwaWeight : REAL ;	//Absolutwert SIWAREX ohne Nullpunktverschiebung
  spare1 : ARRAY  [1 .. 6 ] OF INT ;
  GrossWeight : REAL ;	//Bruttogewicht
  TareWeight : REAL ;	//Tarierspeicher
  NetWeight : REAL ;	//Nettogewicht
  spare2 : ARRAY  [1 .. 4 ] OF INT ;
  SP : STRUCT
   Range : REAL ;	//Scale range
   zero_val : REAL ;	//Zero value
   empty_val : REAL ;	//empty value
   empty_time : INT ;	//empty time
   step_time : INT ;	//step_time
   DosiControlTime : INT ;	//Time for dosing control
  END_STRUCT ;
  PW_IN : STRUCT 	//Aktuelle Prozesswerte
   KoByte : STRUCT
    NV_1 : BOOL ;
    Befehl_ausgefuehrt : BOOL ;	//Siwarex hat den Befehl empfangen (BI)
    LifeBit : BOOL ;	//LB
    Neustart : BOOL ;	//NEUST
    SyncErr : BOOL ;
    WKGN_Bit0 : BOOL ;
    WKGN_Bit1 : BOOL ;
    WKGN_Bit2 : BOOL ;
   END_STRUCT ;
   Zykluszaehler : BYTE ;	//Zykluszähler
   SyncErrCode : BYTE ;	//synchrone Fehlerinfo (Fehlercode)
   AsyncErr : STRUCT 	//asynchrone Fehlerinfo (Bitweise)
    RAM : BOOL ;	//Neuanlauf wegen RAM-Fehler
    Watchdog : BOOL ;	//Neuanlauf wegen Watchdogfehler
    Programm : BOOL ;	//Neuanlauf wegen Programmfehler
    ueberlaufGewicht : BOOL ;	//Zahlerüberlauf bei Gewichtsberechnung
    Parameter : BOOL ;	//Parameterfehler
    Messbereich : BOOL ;	//AD-Wandler an Messbereichsgrenze
    Drahtbruch : BOOL ;	//Mindestspannung an Sense-Leitung unterschritten
    AD_Wandler : BOOL ;	//AD-Wandlerstörung
   END_STRUCT ;
   Prozesswert : INT ;	//Prozesswert (je nach Auswahl im WKNG)
   Status : STRUCT 	//Status
    Schreibschutz : BOOL ;	//Stellung des Schreibschutzschalters (0=AUS 1=EIN)
    MinWB : BOOL ;	//Min.Wägebereich ist unterschritten
    NV_1 : BOOL ;
    NV_2 : BOOL ;
    NV_3 : BOOL ;
    NV_4 : BOOL ;
    NV_5 : BOOL ;
    BaugruppenErr : BOOL ;	//globale Baugruppenstörung
    GW1 : BOOL ;	//Grenzwert 1 hat angesprochen
    GW2 : BOOL ;	//Grenzwert 2 hat angesprochen
    TaraWaage : BOOL ;	//Waage tariert (Taraspeicher belget)
    TaraExt : BOOL ;	//Taraspeicher mit ext. Vorgabewert belegt
    Max_9E : BOOL ;	//Brutto-Wägebereich mehr als 9 Anzeigeschritte über- oder unterschritten
    _1_4dZero : BOOL ;	//Brutto kleiner +/- 0,25e
    Stillstand : BOOL ;	//Stillstand liegt vor
    Justiert : BOOL ;	//Waage justiert
   END_STRUCT ;
  END_STRUCT ;
  PW_OUT : STRUCT
   KoByte : STRUCT
    NV_B0 : BOOL ;
    BefAusfuehren : BOOL ;	//BIQ
    Quitt_LifeBit : BOOL ;	//LBQ
    Quitt_Neustart : BOOL ;	//Neustart bestätigen (NEUSTQ)
    NV_B4 : BOOL ;
    WKGN_Bit0 : BOOL ;
    WKGN_Bit1 : BOOL ;
    WKGN_Bit2 : BOOL ;
   END_STRUCT ;
   BefNummer : BYTE ;
   Ext_Taravorgabe : INT ;
   NV_Byte4 : BYTE ;	//Nicht verwendet
   NV_Byte5 : BYTE ;	//Nicht verwendet
   NV_Byte6 : BYTE ;	//Nicht verwendet
   NV_Byte7 : BYTE ;	//Nicht verwendet
  END_STRUCT ;
  s_JUST_DAT : STRUCT 	//DR3: Calibration parameters
   w_CALIB_DIGITS0 : WORD ;	//Calibration digits for 0
   w_CALIB_DIGITS1 : WORD  := W#16#EA60;	//Calibration digits for 1
   w_CALIB_DIGITS2 : WORD ;	//Calibration digits for 2
   i_CALIB_WEIGHT1 : INT  := 2000;	//Calibration weight for 1
   i_CALIB_WEIGHT2 : INT ;	//Calibration weight for 2
   b_SIGNAL_RANGE : BYTE  := B#16#2;	//Input range (1=1mV/v, 2=2mV/V, 4=4mV/V)
   b_FILT_TYPE : BYTE ;	//Filter type signal filter (only 0 allowed)
   b_FILT_FREQ : BYTE  := B#16#4;	//Filter low pass frequency
   b_FILT_DEPTH : BYTE  := B#16#F;	//Filter depth of average value filter (0...FF)
   s_SCALE_ID : STRING  [10 ] := 'SIWAREX XX';	//Scale identity
   i_MIN_WR : INT  := 20;	//Minimum for weighing range WR
   i_MAX_WR : INT  := 2000;	//Maximum for weighing range WR
   i_INCREMENT_WR : INT  := 1;	//Digital increment for weighing range
   i_WEIGHT_ST_STILL : INT  := 10;	//Stand still weight
   t_TIME_ST_STILL1 : TIME  := T#1S;	//Stand still time in ms
   b_DEC_POINT : BYTE  := B#16#2;	//Decimal point for remote display
   b_ZERO_NEG_VALUE : BYTE  := B#16#1;	//Zeroing negative range (% of WR)
   b_ZERO_POS_VALUE : BYTE  := B#16#3;	//Zeroing positive range (% of WR)
   b_TARA_MAX : BYTE  := B#16#64;	//Tara range (% of WR)
   i_Reserve : INT ;	//Reserve
   s_LEGAL_TRADE : STRING  [4 ] := '----';	//OIML or no ----
   s_WEGHT_UNIT : STRING  [4 ] := 'kg  ';	//Unit for weight
  END_STRUCT ;
  RDREC_1 : SFB 52;
  WRREC_1 : SFB 53;
  ErrTIMER1_SIWA : SFB 4;	//IEC Timer SFB
  ErrTIMER2_SIWA : SFB 4;	//IEC Timer SFB
  ErrTIMER3_SIWA : SFB 4;	//IEC Timer SFB
  TIMER_Res1 : SFB 4;	//Reserve Timer
  TIMER_Res2 : SFB 4;	//Reserve Timer
  TIMER_Pause : SFB 5;	//Reserve Timer
  TIMER_Res3 : SFB 5;	//Reserve Timer
  CMD_Waage_nullen : BOOL ;	//Bit Waage nullen
  CMD_Res1 : BOOL ;	//Reserve
  CMD_Res2 : BOOL ;	//Bit Allgemeine Parameter schreiben
  CMD_Res3 : BOOL ;	//Bit Befehl an Siwarex ausführen
  CMD_Res4 : BOOL ;	//Bit Befehl an Siwarex ausführen
  CMD_Res5 : BOOL ;	//Bit Befehl an Siwarex ausführen
  CMD_Res6 : BOOL ;	//Bit Befehl an Siwarex ausführen
  CMD_Res7 : BOOL ;	//Bit Befehl an Siwarex ausführen
  REQ_Lese_JustDat : BOOL ;	//SFC ausführen
  REQ_Schreibe_JustDat : BOOL ;	//SFC ausführen
  REQ_Schreibe_Befehl : BOOL ;	//SFC ausführen
  REQ_Res1 : BOOL ;	//Reserve
  REQ_Res2 : BOOL ;	//Reserve
  REQ_Res3 : BOOL ;	//Reserve
  REQ_Res4 : BOOL ;	//SFC ausführen
  REQ_Res5 : BOOL ;	//SFC ausführen
  Urloeschschutz : BOOL ;	//Dieses Bit dient dazu um herauszufiltern ob die CPU urgelöscht wurde
  Simulation : BOOL ;	//Simulationsbetrieb !! Waage ist außer Funktion
  FP_Sim : BOOL ;	//Flankenmerker positive Flanke
  FN_Sim : BOOL ;	//Flankenmerker negative Flanke
  SIM_Wert : WORD ;	//Gewichtswert für die Simulation in [g] (max. 65500g)
  SELECT_PROC_VAL : INT ;
  Nullstellwert : WORD ;	//Nullwert der Waage
  Zykluszaehler_OldVal : INT ;
  RET_VAL_JustDat_lesen : DWORD ;	//Rückgabewert SFC Justagedaten lesen
  RET_VAL_JustDat_schrei : DWORD ;	//Rückgabewert SFC Justagedaten schreiben
  Letzter_SFB_RDErrCode : DWORD ;
  Letzter_SFB_WDErrCode : DWORD ;
  SynchronErrCode : INT ;	//Fehlercode
END_VAR
VAR_TEMP
  T_permanent_0 : BOOL ;	//Dauer 0
  T_permanent_1 : BOOL ;	//Dauer 1
  T_DWORD_ADR : DWORD ;	//Siwarex Baugruppenadresse im DWord-Format
  T_BUSY1 : BOOL ;	//SFB ist beschäftigt
  T_BUSY2 : BOOL ;	//SFB ist beschäftigt
  T_Komma_Fak : REAL ;	//Faktor für die Nachkommastelle
  T_Digit_kg : REAL ;	//Digits pro kg
  T_ToggelMesswert : BOOL ;	//Nach jeden neuen Messwert invertiert die Siwarex dieses Bit
  T_Ptr_KoByte : DINT ;
  T_Ptr_Zykluszaehler : DINT ;
  T_Ptr_SyncErr : DINT ;
  T_Ptr_AsyncErr : DINT ;
  T_Ptr_PW : DINT ;
  T_Ptr_Status : DINT ;
  T_Ptr_PW_OUT : DINT ;
  T_Komma : STRUCT
   Komma1 : BOOL ;
   Komma2 : BOOL ;
   Komma3 : BOOL ;
   NV_1 : BOOL ;
   NV_2 : BOOL ;
   NV_3 : BOOL ;
   NV_4 : BOOL ;
   NV_5 : BOOL ;
  END_STRUCT ;
END_VAR
BEGIN
NETWORK
TITLE = Signal permanent1 und permanent0
      CLR;
      =     #T_permanent_0;
      SET;
      =     #T_permanent_1;
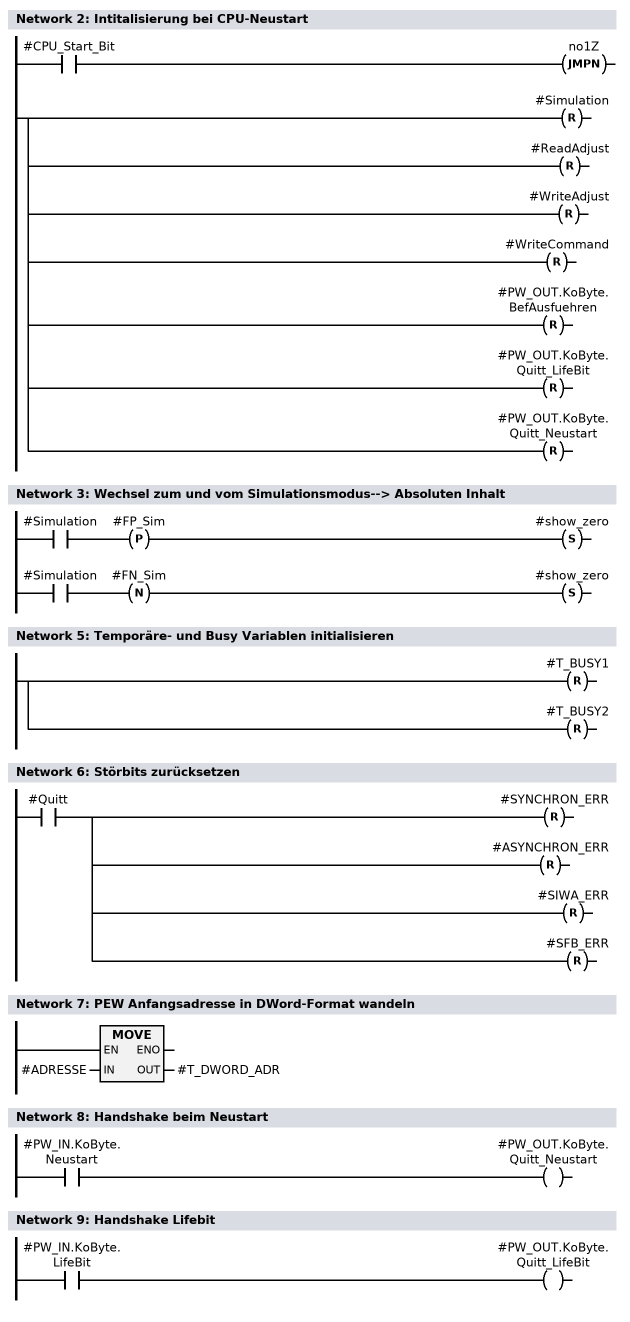
NETWORK
TITLE = Intitalisierung bei CPU-Neustart
//    --------------------------------
      A     #CPU_Start_Bit;
      JCN   no1Z;
      SET;
      R     #Simulation;
      R     #ReadAdjust;
      R     #WriteAdjust;
      R     #WriteCommand;
      R     #PW_OUT.KoByte.BefAusfuehren;
      R     #PW_OUT.KoByte.Quitt_LifeBit;
      R     #PW_OUT.KoByte.Quitt_Neustart;
no1Z: NOP   0;
//    --------------------------------
NETWORK
TITLE = Wechsel zum und vom Simulationsmodus--> Absoluten Inhalt
      A     #Simulation;
      FP    #FP_Sim;
      S     #show_zero;
      A     #Simulation;
      FN    #FN_Sim;
      S     #show_zero;
NETWORK
TITLE = Peripheriedaten in statischen Datenbereich schreiben
      L     P##PW_IN;	//Adresspointer laden
      L     P#0.0;	//Offset von 0 addieren (KoByte)
      +D;
      T     #T_Ptr_KoByte;
      L     P#2.0;	//Offset von 2 addieren (Zykluszaehler)
      +D;
      T     #T_Ptr_Zykluszaehler;
      L     P#1.0;	//Offset von 1 addieren (SyncErrCode)
      +D;
      T     #T_Ptr_SyncErr;
      L     P#1.0;	//Offset von 1 addieren (AsyncErr)
      +D;
      T     #T_Ptr_AsyncErr;
      L     P#2.0;	//Offset von 2 addieren (Prozesswert)
      +D;
      T     #T_Ptr_PW;
      L     P#2.0;	//Offset von 2 addieren (Status)
      +D;
      T     #T_Ptr_Status;
      L     #ADRESSE;	//PEW-Adresse laden
      SLW   3;	//Pointer bilden
      LAR1;
      L     PIB [AR1,P#0.0];	//Peripheriebereich in Statische Daten schreiben
      T     DIB [#T_Ptr_KoByte];
      L     PIB [AR1,P#1.0];
      T     DIB [#T_Ptr_Zykluszaehler];
      L     PIB [AR1,P#2.0];
      T     DIB [#T_Ptr_SyncErr];
      L     PIB [AR1,P#3.0];
      T     DIB [#T_Ptr_AsyncErr];
      L     PIW [AR1,P#4.0];
      A     #Simulation;
      JCN   noSM;
      L     #SIM_Wert;	//Wenn Simulationsbit = 1, dann nehme SIM_Wert als Prozesswert
noSM: T     DIW [#T_Ptr_PW];
      L     PIW [AR1,P#6.0];
      T     DIW [#T_Ptr_Status];
NETWORK
TITLE = Temporäre- und Busy Variablen initialisieren
      SET;
      R     #T_BUSY1;
      R     #T_BUSY2;
NETWORK
TITLE = Störbits zurücksetzen
      A     #Quitt;
      R     #SYNCHRON_ERR;
      R     #ASYNCHRON_ERR;
      R     #SIWA_ERR;
      R     #SFB_ERR;
NETWORK
TITLE = PEW Anfangsadresse in DWord-Format wandeln
      L     #ADRESSE;
      T     #T_DWORD_ADR;
NETWORK
TITLE = Handshake beim Neustart
      A     #PW_IN.KoByte.Neustart;
      =     #PW_OUT.KoByte.Quitt_Neustart;
NETWORK
TITLE = Handshake Lifebit
      A     #PW_IN.KoByte.LifeBit;
      =     #PW_OUT.KoByte.Quitt_LifeBit;
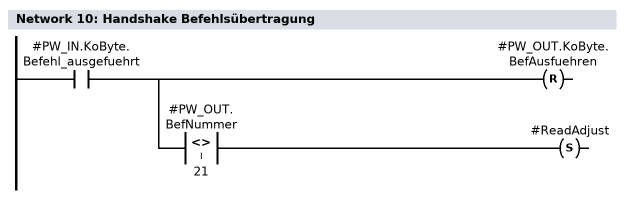
NETWORK
TITLE = Handshake Befehlsübertragung
      A     #PW_IN.KoByte.Befehl_ausgefuehrt;
      =     L 48.0;
      A     L 48.0;
      BLD   102;
      R     #PW_OUT.KoByte.BefAusfuehren;
      A     L 48.0;
      A(;
      L     #PW_OUT.BefNummer;
      L     21;
      <>I;
      );
      S     #ReadAdjust;
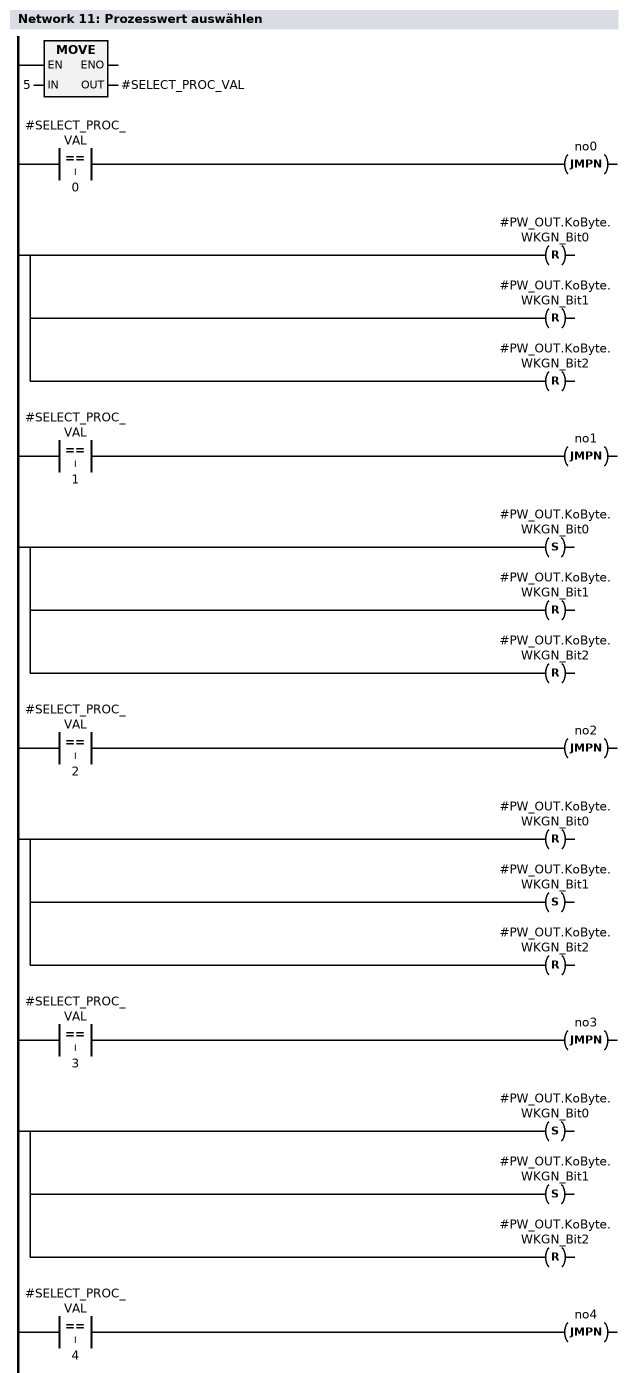
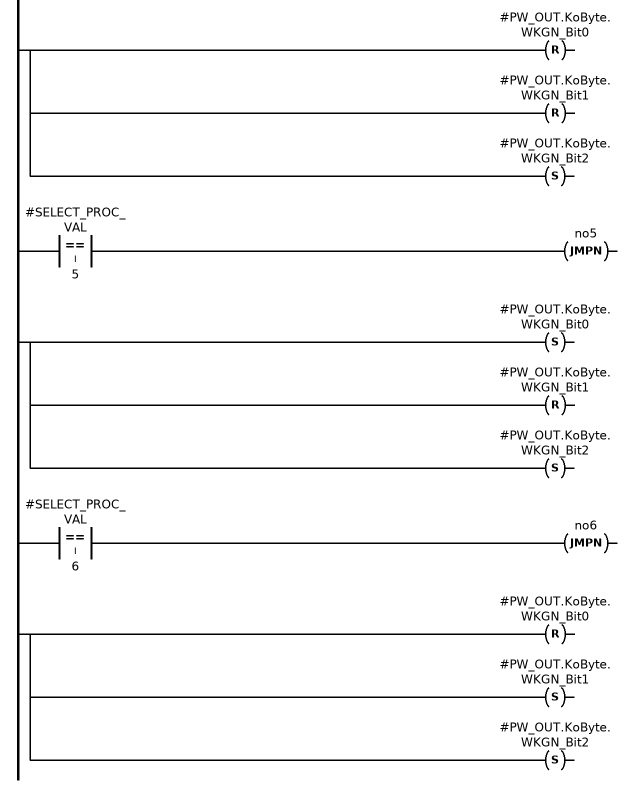
NETWORK
TITLE = Prozesswert auswählen
//0
//B / N-Gewicht (Default)
//Gewicht (je nach Status-Bit SF_NETTO)
//1
//Tara-Gewicht
//Tarawert
//2
//Brutto-Prozesswert
//Brutto
//3
//Netto-Prozesswert
//Netto
//4
//Tara-Prozesswert
//Tara
//5
//gefilterter Roh-Digitwert
//Gefilterter Roh-Digitwert
//6
//ungefilterter Roh-Digitwert
//Ungefilterter Roh-Digitwert
//7
//---
//frei (kein Fehler -> als Wert wird 0 geliefert)
      L     5;	//gefilterter Roh-Digitwert fest auswählen
      T     #SELECT_PROC_VAL;
//    --------------- B / N-Gewicht ------------------
      L     #SELECT_PROC_VAL;
      L     0;
      ==I;
      JCN   no0;
      SET;
      R     #PW_OUT.KoByte.WKGN_Bit0;
      R     #PW_OUT.KoByte.WKGN_Bit1;
      R     #PW_OUT.KoByte.WKGN_Bit2;
no0:  NOP   0;
//    --------------- Tara-Gewicht ------------------
      L     #SELECT_PROC_VAL;
      L     1;
      ==I;
      JCN   no1;
      SET;
      S     #PW_OUT.KoByte.WKGN_Bit0;
      R     #PW_OUT.KoByte.WKGN_Bit1;
      R     #PW_OUT.KoByte.WKGN_Bit2;
no1:  NOP   0;
//    --------------- Brutto-Prozesswert ------------------
      L     #SELECT_PROC_VAL;
      L     2;
      ==I;
      JCN   no2;
      SET;
      R     #PW_OUT.KoByte.WKGN_Bit0;
      S     #PW_OUT.KoByte.WKGN_Bit1;
      R     #PW_OUT.KoByte.WKGN_Bit2;
no2:  NOP   0;
//    --------------- Netto-Prozesswert ------------------
      L     #SELECT_PROC_VAL;
      L     3;
      ==I;
      JCN   no3;
      SET;
      S     #PW_OUT.KoByte.WKGN_Bit0;
      S     #PW_OUT.KoByte.WKGN_Bit1;
      R     #PW_OUT.KoByte.WKGN_Bit2;
no3:  NOP   0;
//    --------------- Tara-Prozesswert ------------------
      L     #SELECT_PROC_VAL;
      L     4;
      ==I;
      JCN   no4;
      SET;
      R     #PW_OUT.KoByte.WKGN_Bit0;
      R     #PW_OUT.KoByte.WKGN_Bit1;
      S     #PW_OUT.KoByte.WKGN_Bit2;
no4:  NOP   0;
//    --------------- gefilterter Roh-Digitwert ------------------
      L     #SELECT_PROC_VAL;
      L     5;
      ==I;
      JCN   no5;
      SET;
      S     #PW_OUT.KoByte.WKGN_Bit0;
      R     #PW_OUT.KoByte.WKGN_Bit1;
      S     #PW_OUT.KoByte.WKGN_Bit2;
no5:  NOP   0;
//    --------------- ungefilterter Roh-Digitwert ------------------
      L     #SELECT_PROC_VAL;
      L     6;
      ==I;
      JCN   no6;
      SET;
      R     #PW_OUT.KoByte.WKGN_Bit0;
      S     #PW_OUT.KoByte.WKGN_Bit1;
      S     #PW_OUT.KoByte.WKGN_Bit2;
no6:  NOP   0;
NETWORK
TITLE = Justagedaten lesen (von SIWAREX zur CPU)
//  ######################################################################################################
//  #   Wenn sich die CPU aus irgend einem Grund urlöscht oder vom Programmierer urgelöscht wird, dann   #
//  #   werden die Justagedaten von der Siwarex in die CPU übertragen. Dies geschieht aber nur,          #
//  #   wenn die Waage bereits justiert war und die CPU gerade hochläuft.                                #
//  ######################################################################################################
      A     #PW_IN.Status.Justiert;
      A     #ANLAUFTIMER;
      AN    #Urloeschschutz;	//wenn dieses Bit den Wert 0 hat, wurde die CPU urgelöscht (Startwert=0)
      S     #ReadAdjust;
//    ---------------------------------
      A     #ReadAdjust;	//Dieses Bit wird entweder eine Zeile oberhalb oder in der VISU gesetzt
      A     #KAS_SIWAREX;
      AN    #BUSY;
      AN    #REQ_Schreibe_JustDat;
      AN    #REQ_Schreibe_Befehl;
      =     #REQ_Lese_JustDat;
//    ---------------------------------
      BLD   16;
      =     L 55.0;
      L     DINO;
      T     LW 53;
      CDB;
      OPN   DI [LW 53];
      TAR2  LD 49;
      A     DBX [AR2,P#403.0];
      =     #RDREC_1.REQ;
      L     #T_DWORD_ADR;
      T     #RDREC_1.ID;
//    ---------------------------------
//----- Wenn der SFB ohne Fehler abgearbeitet wurde wird die Leseanforderung wieder zurückgesetzt -----
      L     3;
      T     #RDREC_1.INDEX;
      L     56;
      T     #RDREC_1.MLEN;	//kein Fehler
      L     W#16#1002;
      T     DIW [AR2,P#212.0];
      L     56;
      T     DIW [AR2,P#214.0];	//nur hier wird das Urlöschschutzbit gesetzt
      L     DBNO;
      T     DIW [AR2,P#216.0];	//Schnittstelle anpassen
      +AR2  P#138.0;	//neu 
      TAR2;	//alt
      LAR2  LD 49;	//neu
      T     DID [AR2,P#218.0];	//alt
      +AR2  P#194.0;
      UC    SFB 52;
      LAR2  LD 49;
      A     #RDREC_1.BUSY;
      =     #T_BUSY1;
      L     #RDREC_1.STATUS;
      T     DBD [AR2,P#414.0];
      CDB;
      BLD   17;
      A     #ReadAdjust;
      A(;
      L     #RET_VAL_JustDat_lesen;
      L     0;
      ==D;
      );
      R     #ReadAdjust;
      S     #Urloeschschutz;
      S     #show_zero;
      JCN   noRD;
      L     #s_JUST_DAT.w_CALIB_DIGITS1;
      T     #AdjustDatas.Digit1;
      L     #s_JUST_DAT.i_CALIB_WEIGHT1;
      T     #AdjustDatas.AdjustWeight;
noRD: NOP   0;
NETWORK
TITLE = Faktor für die Kommastelle berechnen
//Bits:
//Komma1  Komma2  Komma3
//
//0       0       0    Kommastelle 0
//0       0       1    Kommastelle 1
//0       1       0    Kommastelle 2
//0       1       1    Kommastelle 3
//1       0       0    Kommastelle 4
//1       0       1    Kommastelle 5
//
      L     P##T_Komma;	//Adresspointer laden
      L     P#0.0;	//Offset von 0 addieren
      +D;
      LAR1;
      L     #s_JUST_DAT.b_DEC_POINT;
      T     LB [AR1,P#0.0];	//Temp.T_Komma
//---------------------------------------------
      L     1.000000e+00;	//1
      AN    #T_Komma.Komma1;
      JC    KOM2;
      L     1.000000e+01;	//10
      *R;
KOM2: AN    #T_Komma.Komma2;
      JC    KOM3;
      L     1.000000e+02;	//100
      *R;
KOM3: AN    #T_Komma.Komma3;
      JC    KOMe;
      L     1.000000e+04;	//10000
      *R;
KOMe: T     #T_Komma_Fak;	//Faktor für die Kommaverschiebung
NETWORK
TITLE = Siwarexdaten fest beschreiben
      L     0;
      T     #s_JUST_DAT.w_CALIB_DIGITS2;	//Justagepunkt 2 deaktivieren
      T     #s_JUST_DAT.i_CALIB_WEIGHT2;	//Justagepunkt 2 deaktivieren
      T     #s_JUST_DAT.i_MIN_WR;	//Mindestgewicht
//    ---------------------------------
      L     100;
      T     #s_JUST_DAT.b_ZERO_NEG_VALUE;	//Nullfehler in der Siwarex deaktivieren
      T     #s_JUST_DAT.b_ZERO_POS_VALUE;	//Nullfehler in der Siwarex deaktivieren
      T     #s_JUST_DAT.b_TARA_MAX;	//Maximalwert zum Tarieren in %
//    ---------------------------------
      L     1;
      T     #s_JUST_DAT.i_INCREMENT_WR;	//Ziffernschritt auf 1 setzen
      T     #s_JUST_DAT.t_TIME_ST_STILL1;	//Stillstand in der Siwarex deaktivieren
//    ---------------------------------
      L     #s_JUST_DAT.i_MAX_WR;
      L     32767;
      <>I;
      JCN   J0ok;
      L     #s_JUST_DAT.i_MAX_WR;
      L     1;
      -I;
      JP    WTOk;
      L     1;
WTOk: T     #s_JUST_DAT.i_WEIGHT_ST_STILL;
J0ok: NOP   0;
//    ---------------------------------
      A(;
      L     #s_JUST_DAT.i_MAX_WR;
      L     32767;
      ==I;
      );
      A(;
      L     #s_JUST_DAT.i_WEIGHT_ST_STILL;
      L     32767;
      <>I;
      );
      JCN   noTS;
      L     32767;
      T     #s_JUST_DAT.i_WEIGHT_ST_STILL;	//Stillstand in der Siwarex deaktivieren
noTS: NOP   0;
NETWORK
TITLE = Justagedaten schreiben (von CPU in die SIWAREX)
//  #######################################################################################################
//  #     Wenn die Siwarex defekt ist und eine neue (jungfräuliche) Siwarex gesteckt wird, werden die     #
//  #     Justagedaten automatisch beim hochlaufen der CPU von der Steuerung in die Siwarex übertragen.   #                         #
//  #     Somit ist die Siwarex justiert und einsatzbereit. (Austausch der Siwarex)                       #
//  #######################################################################################################      
      AN    #PW_IN.Status.Justiert;	//darum funktioniert das nur bei Jungfräulichkeit(Werkseinstellung)
      A     #ANLAUFTIMER;
      A     #Urloeschschutz;
      S     #WriteAdjust;
//    ---------------------------------
      A     #WriteAdjust;	//Dieses Bit wird entweder eine Zeile oberhalb oder in der VISU gesetzt
      A     #KAS_SIWAREX;
      AN    #BUSY;
      AN    #REQ_Lese_JustDat;
      AN    #REQ_Schreibe_Befehl;
      =     #REQ_Schreibe_JustDat;
//    ---------------------------------
      A     #REQ_Schreibe_JustDat;	//Schnittstelle anpassen
      JCN   noWD;
      L     #AdjustDatas.Digit1;	//alt
      T     #s_JUST_DAT.w_CALIB_DIGITS1;	//neu
      L     #AdjustDatas.AdjustWeight;	//alt
      T     #s_JUST_DAT.i_CALIB_WEIGHT1;	//neu
      L     32767;
      T     #s_JUST_DAT.i_MAX_WR;	//Wägebereich in der Siwarex deaktivieren
noWD: NOP   0;
//    ---------------------------------
      BLD   16;
      =     L 55.0;
      L     DINO;
      T     LW 53;
      CDB;
      OPN   DI [LW 53];
      TAR2  LD 49;
      A     DBX [AR2,P#403.1];
      =     #WRREC_1.REQ;
      L     #T_DWORD_ADR;
//    ---------------------------------
//----- Wenn der SFB ohne Fehler abgearbeitet wurde wird der Schreibeauftrag wieder zurückgesetzt -----
      T     #WRREC_1.ID;
      L     3;
      T     #WRREC_1.INDEX;
      L     56;	//kein Fehler
      T     #WRREC_1.LEN;
      L     W#16#1002;
      T     DIW [AR2,P#238.0];
      L     56;
      T     DIW [AR2,P#240.0];
      L     DBNO;
      T     DIW [AR2,P#242.0];
      +AR2  P#138.0;
      TAR2;
      LAR2  LD 49;
      T     DID [AR2,P#244.0];
      +AR2  P#222.0;
      UC    SFB 53;
      LAR2  LD 49;
      A     #WRREC_1.BUSY;
      =     #T_BUSY2;
      L     #WRREC_1.STATUS;
      T     DBD [AR2,P#418.0];
      CDB;
      BLD   17;
      A     #WriteAdjust;
      A(;
      L     #RET_VAL_JustDat_schrei;
      L     0;
      ==D;
      );
      R     #WriteAdjust;
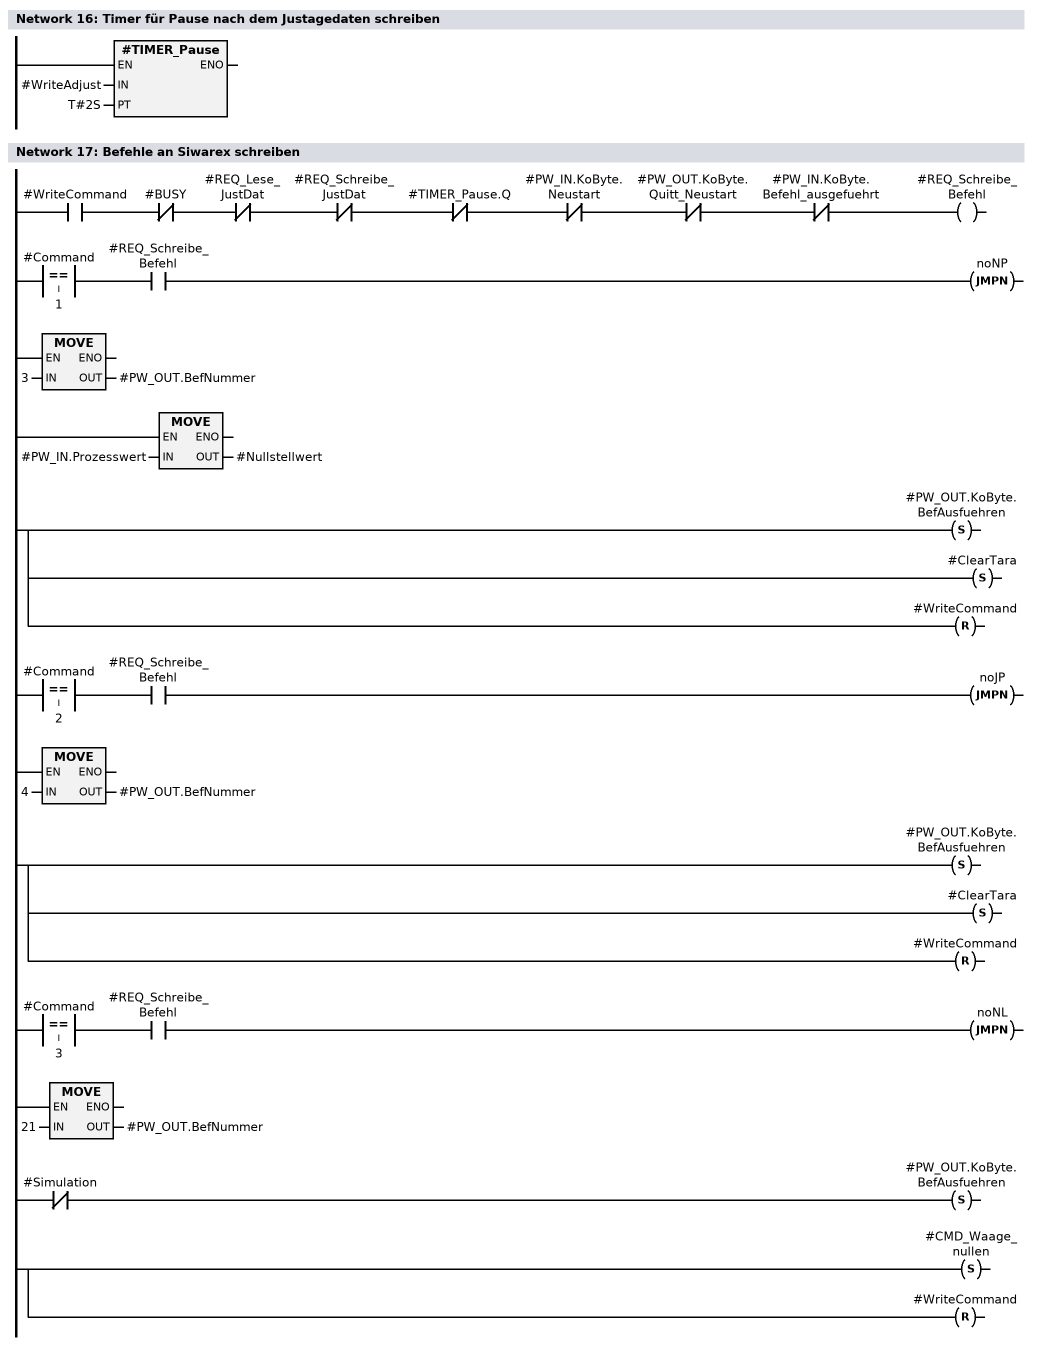
NETWORK
TITLE = Timer für Pause nach dem Justagedaten schreiben
//
//Nach dem Justagedaten schreiben muss eine Pause von 2sek sein, bevor Befehle
//verarbeitet werden können
//
      CALL  #TIMER_Pause (
           IN                       := #WriteAdjust,
           PT                       := T#2S);
NETWORK
TITLE = Befehle an Siwarex schreiben
//1
//DS4 im Flash sichern
//Grenzwertparameter im Flash sichern (DS4)
//2
//DS26 im Flash sichern
//Tara- und Nullstellwert im Flash sichern (DS26)
//3
//Justagebefehl Nullpunkt gültig
//Befehl Nullpunkt gültig (aktiviert den Justierbetrieb)
//Ausführbar wenn kein Schreibschutz (Drahtbrücke 1-5)
//4
//Justagebefehl Justagegewicht 1 gültig
//Der erste Justagepunkt wird durch das Eichgewicht bestimmt.
//Ausführbar wenn kein Schreibschutz (Drahtbrücke 1-5)
//5
//Justagebefehl Justagegewicht 2 gültig
//Der zweite Justagepunkt wird durch das zweite Eichgewicht bestimmt.
//Ausführbar wenn kein Schreibschutz (Drahtbrücke 1-5)
//8
//Alle Datensätze mit Defaultwerten besetzen
//Alle Parameter werden auf den Zustand ab Werk vorbesetzt.
//Ausführbar wenn kein Schreibschutz (Drahtbrücke 1-5)
//15
//Kennlinienverschiebung
//Der Befehl verschiebt die gesamte Kennlinie (die Justagepunkte) so, dass der 
//aktuelle gefilterte Digit-Wert aus dem ADC zu einem neuen Nullpunkt wird. 
//Ergibt 
//sich bei der Verschiebung ein unzulässiger Digit-Wert für einen Justagepunkt, 
//so 
//wird der Befehl abgewiesen.
//Ausführbar wenn kein Schreibschutz (Drahtbrücke 1-5)
//21
//Waage Nullstellen
//Das aktuelle Gewicht wird zu Null gesetzt. Im eichfähigen Betrieb („OIML“) nur 
//eingeschränkt (z.B. –1%, +3%) um den Nullpunkt möglich. Gleichzeitig wird das 
//Taragewicht gelöscht.
//22
//Tarieren
//Das aktuelle Gewicht wird zu Null gesetzt, gleichzeitig wird die 
//Gewichtsanzeige 
//als „Netto“ gekennzeichnet.
//23
//Tara löschen
//Das Taragewicht wird gelöscht. Das aktuelle Gewicht wird angezeigt und 
//Kennzeichnung von „Netto“ auf „Brutto“ umgestellt, die Kennzeichnung „Netto“ 
//und 
//ggf. der Status „Preset-Tara“ wird zurückgesetzt.
//24
//Eingegebenes Tara aus DS15 übernehmen
//Das eingegebene Taragewicht wird als Tara übernommen, gleichzeitig wird die 
//Gewichtsanzeige mit „Netto“ gekennzeichnet und der Status „Preset Tara pT“ 
//gesetzt.
//25
//Erhöhte Auflösung einschalten
//Ausgabe/ Anzeige des eichfähigen Gewichtswertes mit erhöhter Auflösung für 5 
//sec 
//aktivieren.
//26
//Taragewicht aus S7-Steuerbereich übernehmen
//Taravorgabe aus S7-Steuerbereich gültig. Gleichzeitig wird die Gewichtsanzeige 
//mit „Netto“ gekennzeichnet und der Status „Preset Tara pT“ gesetzt
//
      A     #WriteCommand;
      AN    #BUSY;
      AN    #REQ_Lese_JustDat;
      AN    #REQ_Schreibe_JustDat;
      AN    #TIMER_Pause.Q;
      AN    #PW_IN.KoByte.Neustart;
      AN    #PW_OUT.KoByte.Quitt_Neustart;
      AN    #PW_IN.KoByte.Befehl_ausgefuehrt;
      =     #REQ_Schreibe_Befehl;
//    ---------------- Nullpunkt gültig -----------------
      A(;
      L     #Command;
      L     1;
      ==I;
      );
      A     #REQ_Schreibe_Befehl;
      JCN   noNP;
      L     3;
      T     #PW_OUT.BefNummer;
      L     #PW_IN.Prozesswert;
      T     #Nullstellwert;	//Nullstellwert nachführen
      SET;
      S     #PW_OUT.KoByte.BefAusfuehren;
      S     #ClearTara;
      R     #WriteCommand;
noNP: NOP   0;
//    ---------------- Justagepunkt 1 gültig -----------------
      A(;
      L     #Command;
      L     2;
      ==I;
      );
      A     #REQ_Schreibe_Befehl;
      JCN   noJP;
      L     4;
      T     #PW_OUT.BefNummer;
      SET;
      S     #PW_OUT.KoByte.BefAusfuehren;
      S     #ClearTara;
      R     #WriteCommand;
noJP: NOP   0;
//    ---------------- Waage nullen -----------------
      A(;
      L     #Command;
      L     3;
      ==I;
      );
      A     #REQ_Schreibe_Befehl;
      JCN   noNL;
      L     21;
      T     #PW_OUT.BefNummer;
      AN    #Simulation;
      S     #PW_OUT.KoByte.BefAusfuehren;
      SET;
      S     #CMD_Waage_nullen;
      R     #WriteCommand;
noNL: NOP   0;
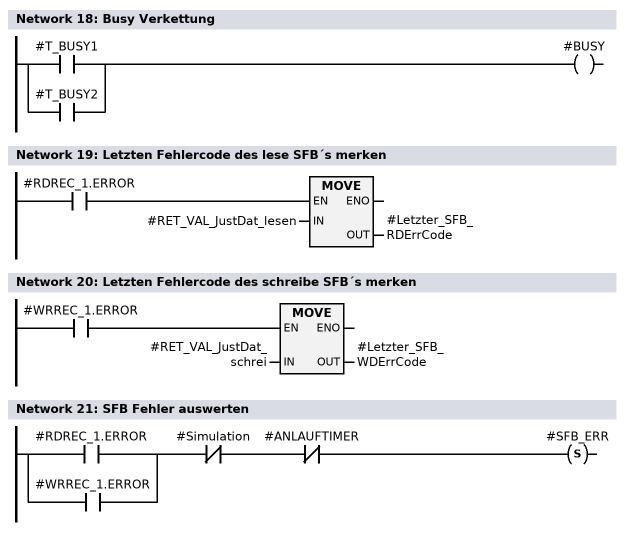
NETWORK
TITLE = Busy Verkettung
//
//                    BUSY = einer der SFB´s ist beschäftigt
//
// Dieses Bit wird benötigt um den anderen Siwarexkanal mitzuteilen das bereits 
//                          ein SFB abgearbeitet wird.
//
      O     #T_BUSY1;
      O     #T_BUSY2;
      =     #BUSY;
NETWORK
TITLE = Letzten Fehlercode des lese SFB´s merken
      A     #RDREC_1.ERROR;
      JNB   _001;
      L     #RET_VAL_JustDat_lesen;
      T     #Letzter_SFB_RDErrCode;
_001: NOP   0;
NETWORK
TITLE = Letzten Fehlercode des schreibe SFB´s merken
      A     #WRREC_1.ERROR;
      JNB   _002;
      L     #RET_VAL_JustDat_schrei;
      T     #Letzter_SFB_WDErrCode;
_002: NOP   0;
NETWORK
TITLE = SFB Fehler auswerten
//  
//   Tritt bei der Bearbeitung eines SFB´s ein Fehler auf wird eine 
//                             Störmeldung gesetzt.
//
      A(;
      O     #RDREC_1.ERROR;
      O     #WRREC_1.ERROR;
      );
      AN    #Simulation;
      AN    #ANLAUFTIMER;
      S     #SFB_ERR;
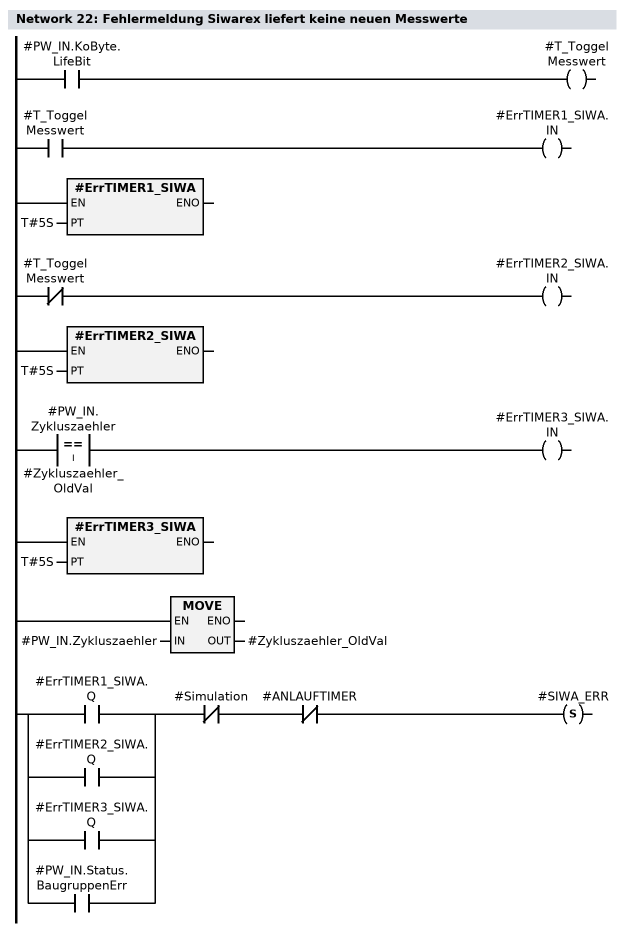
NETWORK
TITLE = Fehlermeldung Siwarex liefert keine neuen Messwerte
//    -----------------------------------------------
      A     #PW_IN.KoByte.LifeBit;
      =     #T_ToggelMesswert;
//    -----------------------------------------------
//    ToggelBit wird nicht mehr zurückgesetzt
      A     #T_ToggelMesswert;
      =     #ErrTIMER1_SIWA.IN;
      CALL  #ErrTIMER1_SIWA (
           PT                       := T#5S);
      AN    #T_ToggelMesswert;
      =     #ErrTIMER2_SIWA.IN;
//    -----------------------------------------------
//    -----------------------------------------------
//    ToggelBit wird nicht mehr gesetzt
      CALL  #ErrTIMER2_SIWA (
           PT                       := T#5S);
      L     #PW_IN.Zykluszaehler;
      L     #Zykluszaehler_OldVal;
      ==I;
      =     #ErrTIMER3_SIWA.IN;
      CALL  #ErrTIMER3_SIWA (
           PT                       := T#5S);
//    -----------------------------------------------
//    -----------------------------------------------
      L     #PW_IN.Zykluszaehler;
      T     #Zykluszaehler_OldVal;
      A(;
      O     #ErrTIMER1_SIWA.Q;
      O     #ErrTIMER2_SIWA.Q;
      O     #ErrTIMER3_SIWA.Q;
      O     #PW_IN.Status.BaugruppenErr;
      );
      AN    #Simulation;
      AN    #ANLAUFTIMER;
      S     #SIWA_ERR;
//    -----------------------------------------------
NETWORK
TITLE = Fehlermeldung Synchronfehler
//
//DIX55.0 ist der "Abstand der Justierpunkte zu klein" der alte Schnittstelle
//
      A     #PW_IN.KoByte.SyncErr;
      AN    #Simulation;
      AN    #ANLAUFTIMER;
      S     #SYNCHRON_ERR;
      A     #SYNCHRON_ERR;
      L     0;
      JCN   noSE;
      L     #PW_IN.SyncErrCode;
noSE: T     #SynchronErrCode;
      O(;
      L     #SynchronErrCode;
      L     85;
      ==I;
      );
      O(;
      L     #SynchronErrCode;
      L     86;
      ==I;
      );
      O(;
      L     #SynchronErrCode;
      L     94;
      ==I;
      );
      =     DIX 55.0;
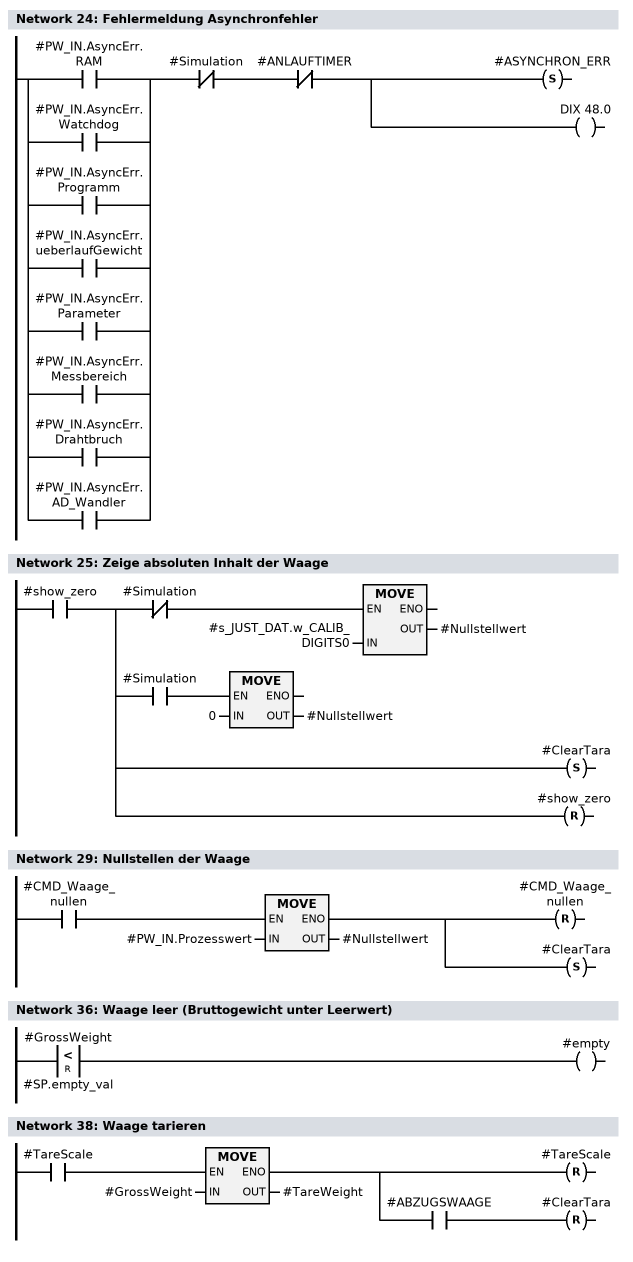
NETWORK
TITLE = Fehlermeldung Asynchronfehler
//
//DIX48.0 ist der Asynchronfehler der alten Schnittstelle
//
      A(;
      O     #PW_IN.AsyncErr.RAM;
      O     #PW_IN.AsyncErr.Watchdog;
      O     #PW_IN.AsyncErr.Programm;
      O     #PW_IN.AsyncErr.ueberlaufGewicht;
      O     #PW_IN.AsyncErr.Parameter;
      O     #PW_IN.AsyncErr.Messbereich;
      O     #PW_IN.AsyncErr.Drahtbruch;
      O     #PW_IN.AsyncErr.AD_Wandler;
      );
      AN    #Simulation;
      AN    #ANLAUFTIMER;
      S     #ASYNCHRON_ERR;
      =     DIX 48.0;
NETWORK
TITLE = Zeige absoluten Inhalt der Waage
      A     #show_zero;
      =     L 49.0;
      A     L 49.0;
      AN    #Simulation;
      JNB   _003;
      L     #s_JUST_DAT.w_CALIB_DIGITS0;
      T     #Nullstellwert;
_003: NOP   0;
      A     L 49.0;
      A     #Simulation;
      JNB   _004;
      L     0;
      T     #Nullstellwert;
_004: NOP   0;
      A     L 49.0;
      BLD   102;
      S     #ClearTara;
      A     L 49.0;
      BLD   102;
      R     #show_zero;
NETWORK
TITLE = Digitwert pro kg berechnen
//
//        Digit 1 - Digit 0
//       -------------------  *   Kommafaktor   =  Digits pro kg
//         Justagegewicht
//
      L     #s_JUST_DAT.w_CALIB_DIGITS1;
      L     #s_JUST_DAT.w_CALIB_DIGITS0;
      -D;
      DTR;
      L     #s_JUST_DAT.i_CALIB_WEIGHT1;
      ITD;
      DTR;
      /R;
      L     #T_Komma_Fak;	//Da Justagegewicht vom Datentyp Integer und die Nachkommastellen aufmultipliziert werden,
      *R;	//muss hier Korrektur gerechnet werden. Darum der Kommafaktor.
      A     #Simulation;
      JCN   Sm03;
      L     1.000000e+03;	// Wenn Bit Simulation = 1, dann entspricht 1000 Digit = 1 kg
Sm03: T     #T_Digit_kg;	// Digits pro kg
NETWORK
TITLE = Berechne Gewichtswert Siwarex ohne Nullpunktverschiebung
//
//        aktueller Digitwert - Digit 0
//       ------------------------------------   =  Absolutgewicht
//                  Digits pro kg
//
      L     #PW_IN.Prozesswert;
      L     #s_JUST_DAT.w_CALIB_DIGITS0;
      -D;
      DTR;
      L     #T_Digit_kg;
      /R;
      A     #Simulation;
      JCN   Sm04;
      L     #PW_IN.Prozesswert;	//Hier nur wenn Bit Simulation = 1
      L     0;
      -D;
      DTR;
      L     #T_Digit_kg;
      /R;
Sm04: T     #SiwaWeight;	//Absolutwert SIWAREX ohne Nullpunktverschiebung
NETWORK
TITLE = Nullwert prüfen
//
//   ############ Absolutgewicht der Waage > Nullwert = Nullfehler ###########
//
      L     #SiwaWeight;
      ABS;	// +/- Richtung wird überprüft
      L     #SP.zero_val;
      >R;
      =     #no_zero;
      A     #no_zero;
      A     #CMD_Waage_nullen;
      R     #CMD_Waage_nullen;
      R     #PW_OUT.KoByte.BefAusfuehren;
NETWORK
TITLE = Nullstellen der Waage
//
//Stillstand wird im FC61 geprüft
//
      A     #CMD_Waage_nullen;
      JNB   _005;
      L     #PW_IN.Prozesswert;
      T     #Nullstellwert;
      SET;
      SAVE;
      CLR;
_005: A     BR;
      R     #CMD_Waage_nullen;
      S     #ClearTara;
NETWORK
TITLE = Bruttowert berechnen
//
//        aktueller Digitwert - Nullstellwert
//       ------------------------------------   =  Bruttowert
//                  Digits pro kg
//
      L     #PW_IN.Prozesswert;
      L     #Nullstellwert;
      -D;
      DTR;
      L     #T_Digit_kg;
      /R;
      T     #GrossWeight;
NETWORK
TITLE = Gewichtswert für Dosierzeit- und Stillstandskontrolle berechnen
      L     #GrossWeight;
      L     #T_Komma_Fak;
      *R;
      RND;
      T     #ActDatas.Gross;
NETWORK
TITLE = Dosierzeitkontrolle
//
//              hier wird kontrolliert ob
//     sich der Gewichtswert der Waage geändert hat
//                 |            |     
//
//     ___________   __________   _____.....usw.
//    |           | |          | |
//    |    -T-    | |    -T-   | |
//    |           | |          | |
//   _|           |_|          |_|
//
      L     #SP.DosiControlTime;
      L     0;
      ==I;
      JC    d_n;	// no Dosing Time control
      A     #dosing;
      JC    dos;
      L     #ActDatas.Gross;
      L     10;
      -I;
      T     #DosiControl_OldVal;
      SET;
      T     LD 49;
      TAK;
      T     LD 53;
      L     #DosiControlTimer;
      T     LW 57;
      L     LD 53;
      L     LD 49;	// time base  1s in highest Nibble
      R     T [LW 57];
      R     #DosiControl;
dos:  T     LD 49;
      TAK;
      T     LD 53;
      L     #DosiControlTimer;
      T     LW 57;
      L     LD 53;
      L     LD 49;
      AN    T [LW 57];	//standstill
      A     #dosing;
      L     #SP.DosiControlTime;
      ITB;
      L     W#16#2000;
      OW;
      T     LD 49;
      TAK;	//new value is old value
      T     LD 53;
      L     #DosiControlTimer;
      T     LW 57;
      L     LD 53;
      L     LD 49;
      SE    T [LW 57];
      NOT;
      JC    d_ex;
      L     #ActDatas.Gross;
      L     #DosiControl_OldVal;
      -I;
      JP    d_p;
      NEGI;
d_p:  L     1;
      >I;
      JC    d_n;
      SET;
      S     #DosiControl;
      JU    d_t;
d_n:  R     #DosiControl;
d_t:  L     #ActDatas.Gross;
      T     #DosiControl_OldVal;
d_ex: NOP   0;
NETWORK
TITLE = Fortschaltezeit
      A     #dosing;
      L     #SP.step_time;
      ITB;
      L     W#16#2000;
      OW;
      T     LD 49;
      TAK;
      T     LD 53;
      L     #StepTimer;
      T     LW 57;
      L     LD 53;
      L     LD 49;
      SF    T [LW 57];
      T     LD 49;
      TAK;
      T     LD 53;
      L     #StepTimer;
      T     LW 57;
      L     LD 53;
      L     LD 49;
      A     T [LW 57];
      =     #StepTime;
NETWORK
TITLE = Stillstand der Waage überprüfen
//
//              hier wird kontrolliert ob
//     sich der Gewichtswert der Waage geändert hat
//                 |            |     
//
//     ___________   __________   _____.....usw.
//    |           | |          | |
//    |    -T-    | |    -T-   | |
//    |           | |          | |
//   _|           |_|          |_|
//
      T     LD 49;
      TAK;	//standstill time
      T     LD 53;
      L     #StillTimer;
      T     LW 57;
      L     LD 53;
      L     LD 49;
      AN    T [LW 57];
      L     S5T#1S;
      T     LD 49;
      TAK;	//standstill
      T     LD 53;
      L     #StillTimer;
      T     LW 57;	//Der Stillstand der Siwarex CS muss hier noch Abgefragt werden, da sie bei nicht Stillstand keine Befehle annimmt
      L     LD 53;
      L     LD 49;
      SE    T [LW 57];
      NOT;	//new value is old value
      JC    s_ex;
      L     #ActDatas.Gross;
      L     #StandStill_OldVal;
      -I;
      JP    s_p;
      NEGI;
s_p:  L     1;
      >I;
      JC    s_n;
      A     #PW_IN.Status.Stillstand;
      S     #Standstill;
      JU    s_t;
s_n:  R     #Standstill;
s_t:  L     #ActDatas.Gross;
      T     #StandStill_OldVal;
s_ex: NOP   0;
NETWORK
TITLE = Überlast
//
//    ##########  Bruttowert > (Wägebereich + 5%) = Waage Überlast  ##########
//
      L     #SP.Range;
      L     1.050000e+00;	//+5%
      *R;
      L     #GrossWeight;
      TAK;
      >R;
      =     #Overload;
NETWORK
TITLE = Waage leer (Bruttogewicht unter Leerwert)
//
//    ##########  Bruttowert < Leerwert der Waage = Waage leer  ##########
//
      L     #GrossWeight;
      L     #SP.empty_val;
      <R;
      =     #empty;
NETWORK
TITLE = Waage Leer und Leerzeit abgelaufen
//
//(Bruttowert < Leerwert der Waage) + Leerzeit abgelaufen = Leerzeit  
//
      A     #empty;
      A     #discharge;
      L     #SP.empty_time;
      ITB;
      L     W#16#2000;
      OW;
      T     LD 49;
      TAK;
      T     LD 53;
      L     #EmptyTimer;
      T     LW 57;
      L     LD 53;
      L     LD 49;
      SD    T [LW 57];
      T     LD 49;
      TAK;
      T     LD 53;
      L     #EmptyTimer;
      T     LW 57;
      L     LD 53;
      L     LD 49;
      A     T [LW 57];
      =     #time_empty;
NETWORK
TITLE = Waage tarieren
//
//Bruttowert in Taraspeicher sichern
//Stillstand wird im Dosierbaustein geprüft
      A     #TareScale;
      JNB   _006;
      L     #GrossWeight;
      T     #TareWeight;
      SET;
      SAVE;
      CLR;
_006: A     BR;
      =     L 49.0;
      A     L 49.0;
      BLD   102;
      R     #TareScale;
      A     L 49.0;
      A     #ABZUGSWAAGE;
      R     #ClearTara;
NETWORK
TITLE = Taraspeicher löschen (Inhalt der Waage anzeigen)
//
//Taraspeicher wird mit Null beschrieben
//
      AN    #ClearTara;
      JC    noIn;
      AN    #ABZUGSWAAGE;
      JC    noAb;
//          --- für Abzugswaage ---
      L     0.000000e+00;
      T     #TareWeight;
      L     #GrossWeight;
      JU    NETT;
//          ----- für Zuwaage -----
noAb: L     0.000000e+00;
      T     #TareWeight;
      SET;
      R     #ClearTara;
noIn: NOP   0;
NETWORK
TITLE = Nettowert berechnen
//
//Formel für Zuwaage:         ##### Bruttowert - Taraspeicher = Nettowert ######
//
//Formel für Abzugswaage:   ### (Taraspeicher - Bruttowert) * -1 = Nettowert ###
//
      L     #GrossWeight;
      L     #TareWeight;
      -R;
      AN    #ABZUGSWAAGE;
      JC    NETT;
//          ----- speziell für Abzugswaage -----
      L     #TareWeight;
      L     #GrossWeight;
      -R;
      AN    #ClearTara;
      JC    NETT;
      L     -1.000000e+00;	//aus negativ mach positiv
      *R;
NETT: T     #NetWeight;
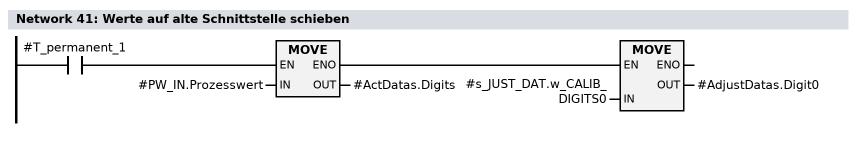
NETWORK
TITLE = Werte auf alte Schnittstelle schieben
      A(;
      A     #T_permanent_1;
      JNB   _007;
      L     #PW_IN.Prozesswert;
      T     #ActDatas.Digits;
      SET;
      SAVE;
      CLR;
_007: A     BR;
      );
      JNB   _008;
      L     #s_JUST_DAT.w_CALIB_DIGITS0;
      T     #AdjustDatas.Digit0;
_008: NOP   0;
NETWORK
TITLE = Ausgangsdaten an die Peripherie schreiben
//    ---------------------------------
      L     P##PW_OUT;	//Adresspointer laden
      L     P#0.0;	//Offset von 0 addieren (KoByte)
      +D;
      T     #T_Ptr_PW_OUT;
//    ---------------------------------
//    ---------------------------------
      L     #ADRESSE;	//PEW-Adresse laden
      SLW   3;	//Pointer bilden
      LAR1;
//    ---------------------------------
      L     DIB [#T_Ptr_PW_OUT];
      T     PQB [AR1,P#0.0];	//Byte 0
//    ---------------------------------
      L     #T_Ptr_PW_OUT;
      L     P#2.0;	//Offset von 2 addieren (BefNummer)
      +D;
      T     #T_Ptr_PW_OUT;
      L     DIB [#T_Ptr_PW_OUT];
      T     PQB [AR1,P#1.0];	//Byte 1
//    ---------------------------------
//Die restlichen Bytes werden nicht verwendent, darum auch nicht in die Peripherie transferiert
END_FUNCTION_BLOCK

FUNCTION FC 1 : VOID
TITLE = Fault indication/horn
VERSION : 0.1
VAR_TEMP
  Stoer : BOOL ;
  ptr : DINT ;
  ctr : DINT ;
  err_sum : DINT ;
  loop_ctr : INT ;
  err_ptr : DINT ;
  quit_ptr : DINT ;
  err_length : INT ;
  quit_length : INT ;
  err_ptr2 : DINT ;
  quit_ptr2 : DINT ;
  err_length2 : INT ;
  quit_length2 : INT ;
  loop_ctr2 : INT ;
END_VAR
BEGIN
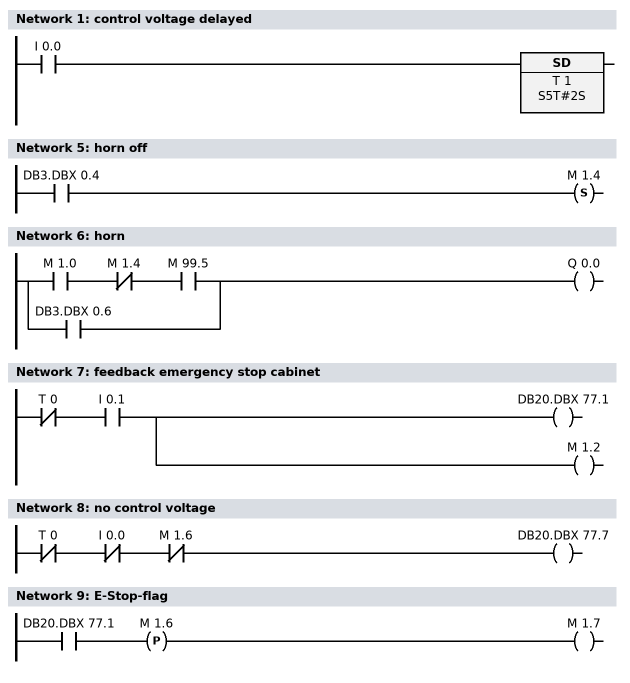
NETWORK
TITLE = control voltage delayed
      A     I 0.0;
      L     S5T#2S;
      SD    T 1;
NETWORK
TITLE = Test on error Gravimet
      OPN   DB 20;
      L     P#72.0;
      T     #ptr;
      L     0;
      T     #err_sum;
      OPN   DB 20;
      L     10;
lp1:  T     #loop_ctr;
      L     DBW [#ptr];
      L     #err_sum;
      +D;
      T     #err_sum;
      L     #ptr;
      L     P#2.0;
      +D;
      T     #ptr;
      L     #loop_ctr;
      LOOP  lp1;
      L     #err_sum;
      L     0;
      <>I;
      =     M 1.0;
      O(;
      A     M 1.0;
      A     M 99.5;
      );
      O     DB3.DBX 0.6;
      =     DB3.DBX 20.2;
NETWORK
TITLE = acknowlege errors Gravimet
      L     P#72.0;
      T     #err_ptr;
      L     P#92.0;
      T     #quit_ptr;
      L     10;
      T     #err_length;
      T     #quit_length;
      OPN   DB 20;
      AN    M 207.7;	//quit
      JC    M014;
      L     #quit_length;	// Anz Worte Quittierbereich
M017: T     #loop_ctr;
      L     DW#16#FFFFFFFF;
      T     DBW [#quit_ptr];
      L     #quit_ptr;
      L     P#2.0;
      +D;
      T     #quit_ptr;
      L     #loop_ctr;
      LOOP  M017;
      JU    M015;
M014: L     10;
M018: T     #loop_ctr;
      L     0;
      T     DBW [#quit_ptr];
      L     #quit_ptr;
      L     P#2.0;
      +D;
      T     #quit_ptr;
      L     #loop_ctr;
      LOOP  M018;
M015: A     M 207.7;
      FN    M 201.5;
      JCN   M016;
      L     10;
M019: T     #loop_ctr;
      L     0;
      T     DBW [#err_ptr];
      L     #err_ptr;
      L     P#2.0;
      +D;
      T     #err_ptr;
      L     #loop_ctr;
      LOOP  M019;
M016: NOP   0;
NETWORK
TITLE = horn off Gravimet
      AN    M 1.0;
      R     M 1.4;
      L     P#72.0;	//  Beginn Fehlerbereich
      T     #ptr;
      L     160;	// Länge Fehlerbereich (BIT)
lp:   T     #ctr;
      OPN   DB 20;
      AN    DBX [#ptr];	// Fehler nicht da
      JC    nerr;
      A     DBX [#ptr];	// Fehler schon gemeldet??
      OPN   DB 19;
      A     DBX [#ptr];
      JC    nego;	// ja
      AN    DBX [#ptr];
      S     DBX [#ptr];	// Fehler gemeldet setzen
      R     M 1.4;	// Hupe einschalten
      JU    nego;
nerr: OPN   DB 19;	// "Fehler gemeldet" löschen
      A     M 0.1;
      R     DBX [#ptr];
nego: L     #ptr;	// nächster Fehler
      INC   1;
      T     #ptr;
      L     #ctr;
      LOOP  lp;
NETWORK
TITLE = horn off
      A     DB3.DBX 0.4;
      S     M 1.4;
NETWORK
TITLE = horn
//ok
      A     M 1.0;
      AN    M 1.4;
      A     M 99.5;
      O     DB3.DBX 0.6;
      =     Q 0.0;
NETWORK
TITLE = feedback emergency stop cabinet
      AN    T 0;
      A     I 0.1;
      =     DB20.DBX 77.1;
      =     M 1.2;
NETWORK
TITLE = no control voltage
      AN    T 0;
      AN    I 0.0;
      AN    M 1.6;
      =     DB20.DBX 77.7;
NETWORK
TITLE = E-Stop-flag
      A     DB20.DBX 77.1;
      FP    M 1.6;
      =     M 1.7;
END_FUNCTION

FUNCTION FC 2 : VOID
TITLE = Automatic run
VERSION : 0.1
VAR_TEMP
  rem_start : BOOL ;
  rem_start_L : BOOL ;
END_VAR
BEGIN
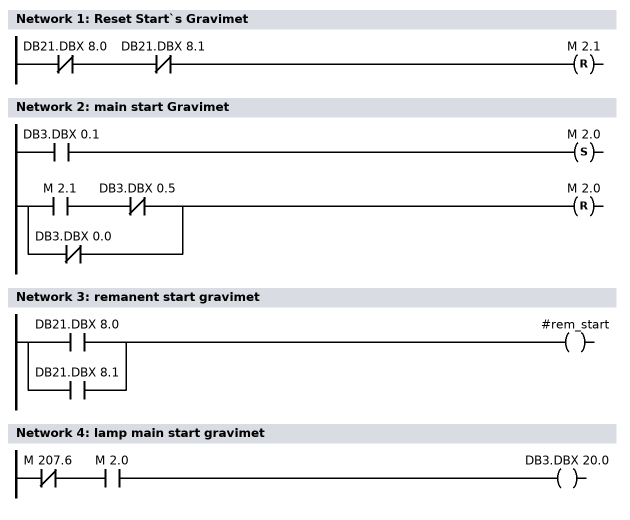
NETWORK
TITLE = Reset Start`s Gravimet
      AN    DB21.DBX 8.0;
      AN    DB21.DBX 8.1;
      R     M 2.1;
NETWORK
TITLE = main start Gravimet
      A     DB3.DBX 0.1;
      S     M 2.0;
      A(;
      A     M 2.1;
      AN    DB3.DBX 0.5;
      ON    DB3.DBX 0.0;
      );
      R     M 2.0;
      NOP   0;
NETWORK
TITLE = remanent start gravimet
      O     DB21.DBX 8.0;
      O     DB21.DBX 8.1;
      =     #rem_start;
NETWORK
TITLE = lamp main start gravimet
      AN    M 207.6;
      A     M 2.0;
      =     DB3.DBX 20.0;
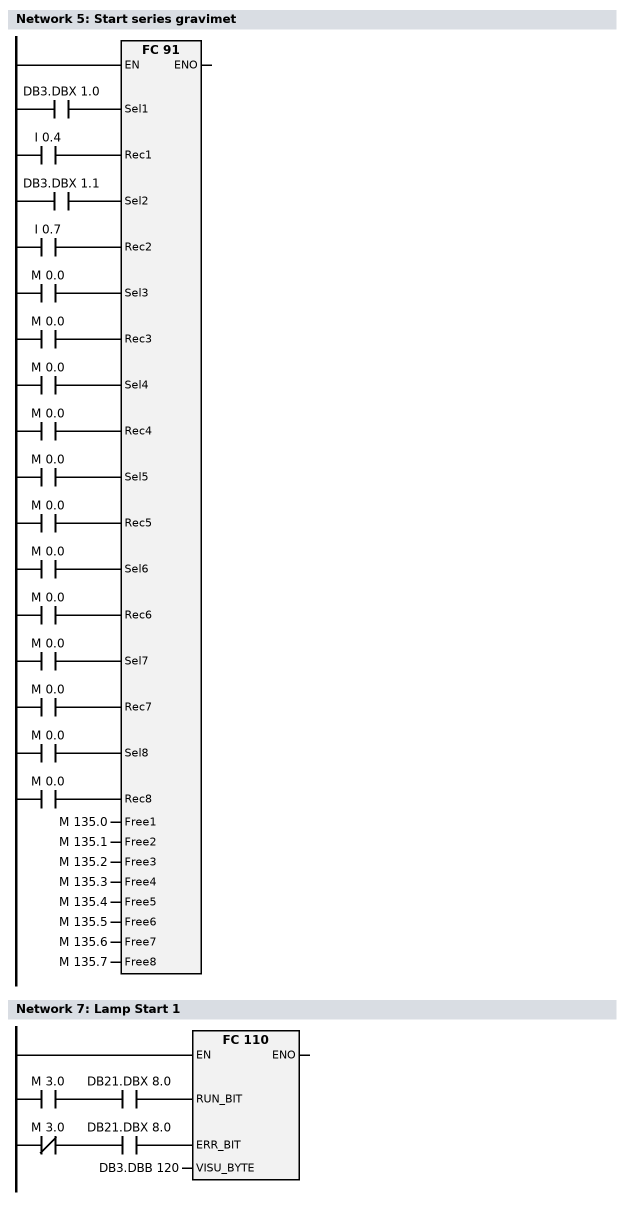
NETWORK
TITLE = Start series gravimet
      A     DB3.DBX 1.0;
      =     L 1.0;
      BLD   103;
      A     I 0.4;
      =     L 1.1;
      BLD   103;
      A     DB3.DBX 1.1;
      =     L 1.2;
      BLD   103;
      A     I 0.7;
      =     L 1.3;
      BLD   103;
      A     M 0.0;
      =     L 1.4;
      BLD   103;
      A     M 0.0;
      =     L 1.5;
      BLD   103;
      A     M 0.0;
      =     L 1.6;
      BLD   103;
      A     M 0.0;
      =     L 1.7;
      BLD   103;
      A     M 0.0;
      =     L 2.0;
      BLD   103;
      A     M 0.0;
      =     L 2.1;
      BLD   103;
      A     M 0.0;
      =     L 2.2;
      BLD   103;
      A     M 0.0;
      =     L 2.3;
      BLD   103;
      A     M 0.0;
      =     L 2.4;
      BLD   103;
      A     M 0.0;
      =     L 2.5;
      BLD   103;
      A     M 0.0;
      =     L 2.6;
      BLD   103;
      A     M 0.0;
      =     L 2.7;
      BLD   103;
      CALL  FC 91 (
           Sel1                     := L 1.0,
           Rec1                     := L 1.1,
           Sel2                     := L 1.2,
           Rec2                     := L 1.3,
           Sel3                     := L 1.4,
           Rec3                     := L 1.5,
           Sel4                     := L 1.6,
           Rec4                     := L 1.7,
           Sel5                     := L 2.0,
           Rec5                     := L 2.1,
           Sel6                     := L 2.2,
           Rec6                     := L 2.3,
           Sel7                     := L 2.4,
           Rec7                     := L 2.5,
           Sel8                     := L 2.6,
           Rec8                     := L 2.7,
           Free1                    := M 135.0,
           Free2                    := M 135.1,
           Free3                    := M 135.2,
           Free4                    := M 135.3,
           Free5                    := M 135.4,
           Free6                    := M 135.5,
           Free7                    := M 135.6,
           Free8                    := M 135.7);
      NOP   0;
NETWORK
TITLE = Start 1
      A(;
      A     M 135.0;
      A     M 2.0;
      S     DB21.DBX 8.0;
      A     M 2.1;
      R     DB21.DBX 8.0;
      A     DB21.DBX 8.0;
      );
      A     M 2.0;
      =     M 3.0;
NETWORK
TITLE = Lamp Start 1
      A     M 3.0;
      A     DB21.DBX 8.0;
      =     L 1.0;
      BLD   103;
      AN    M 3.0;
      A     DB21.DBX 8.0;
      =     L 1.1;
      BLD   103;
      CALL  FC 110 (
           RUN_BIT                  := L 1.0,
           ERR_BIT                  := L 1.1,
           VISU_BYTE                := DB3.DBB 120);
      NOP   0;
NETWORK
TITLE = Start 2
      A(;
      A     M 135.1;
      A     M 2.0;
      S     DB21.DBX 8.1;
      A     M 2.1;
      R     DB21.DBX 8.1;
      A     DB21.DBX 8.1;
      );
      A     M 2.0;
      =     M 3.1;
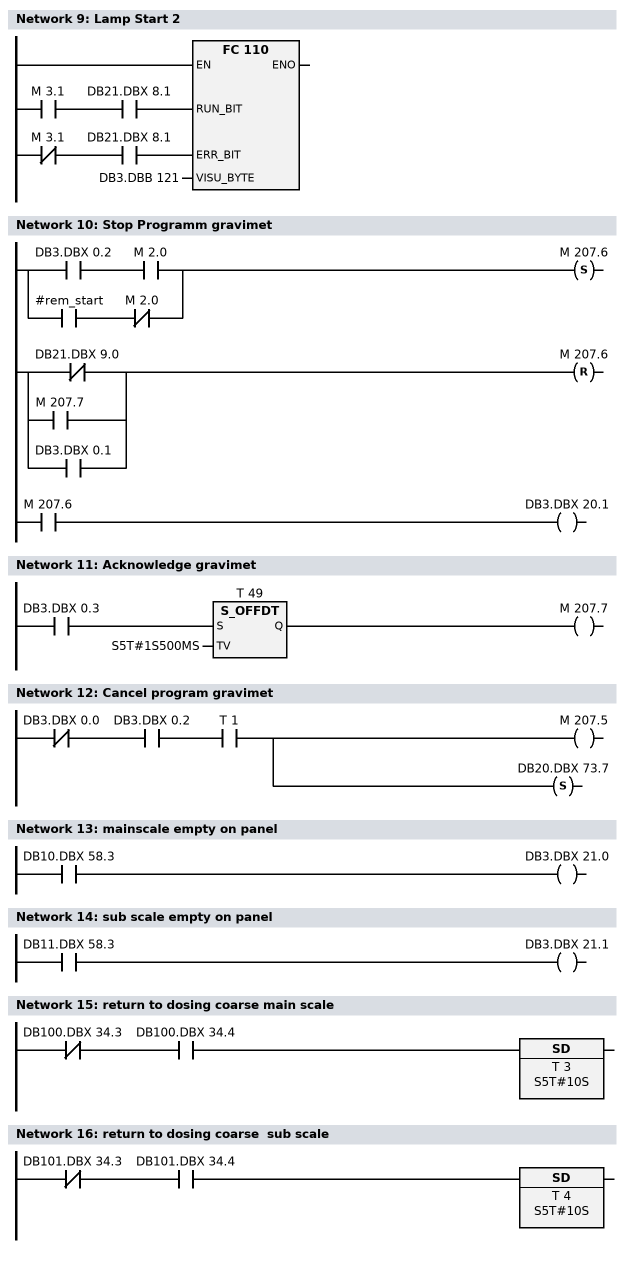
NETWORK
TITLE = Lamp Start 2
      A     M 3.1;
      A     DB21.DBX 8.1;
      =     L 1.0;
      BLD   103;
      AN    M 3.1;
      A     DB21.DBX 8.1;
      =     L 1.1;
      BLD   103;
      CALL  FC 110 (
           RUN_BIT                  := L 1.0,
           ERR_BIT                  := L 1.1,
           VISU_BYTE                := DB3.DBB 121);
      NOP   0;
NETWORK
TITLE = Stop Programm gravimet
      A(;
      A     DB3.DBX 0.2;
      A     M 2.0;
      O;
      A     #rem_start;
      AN    M 2.0;
      );
      S     M 207.6;
      A(;
      ON    DB21.DBX 9.0;
      O     M 207.7;
      O     DB3.DBX 0.1;
      );
      R     M 207.6;
      A     M 207.6;
      =     DB3.DBX 20.1;
NETWORK
TITLE = Acknowledge gravimet
      A     DB3.DBX 0.3;
      L     S5T#1S500MS;
      SF    T 49;
      NOP   0;
      NOP   0;
      NOP   0;
      A     T 49;
      =     M 207.7;
NETWORK
TITLE = Cancel program gravimet
      AN    DB3.DBX 0.0;
      A     DB3.DBX 0.2;
      A     T 1;
      =     M 207.5;
      S     DB20.DBX 73.7;
NETWORK
TITLE = mainscale empty on panel
      A     DB10.DBX 58.3;
      =     DB3.DBX 21.0;
NETWORK
TITLE = sub scale empty on panel
      A     DB11.DBX 58.3;
      =     DB3.DBX 21.1;
NETWORK
TITLE = return to dosing coarse main scale
      AN    DB100.DBX 34.3;
      A     DB100.DBX 34.4;
      L     S5T#10S;
      SD    T 3;
NETWORK
TITLE = return to dosing coarse  sub scale
      AN    DB101.DBX 34.3;
      A     DB101.DBX 34.4;
      L     S5T#10S;
      SD    T 4;
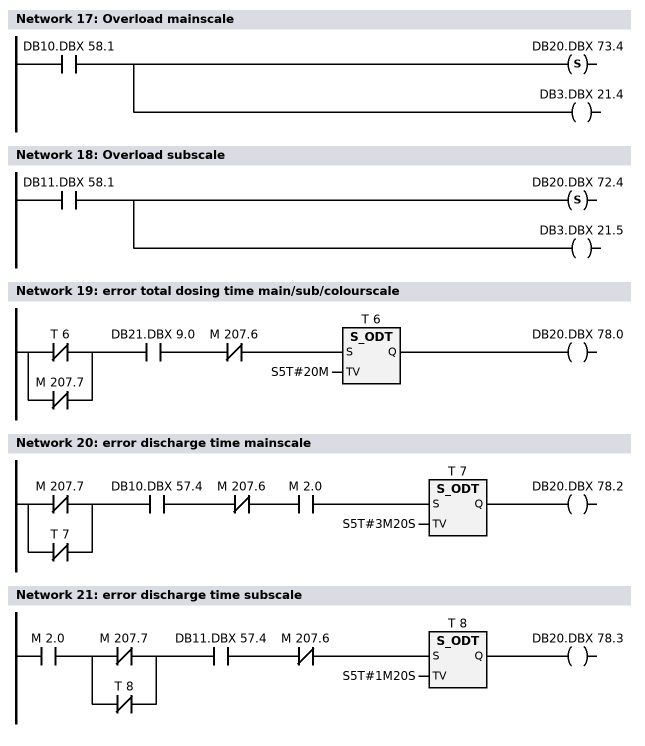
NETWORK
TITLE = Overload mainscale
      A     DB10.DBX 58.1;
      S     DB20.DBX 73.4;
      =     DB3.DBX 21.4;
NETWORK
TITLE = Overload subscale
      A     DB11.DBX 58.1;
      S     DB20.DBX 72.4;
      =     DB3.DBX 21.5;
NETWORK
TITLE = error total dosing time main/sub/colourscale
      A(;
      ON    T 6;
      ON    M 207.7;
      );
      A     DB21.DBX 9.0;
      AN    M 207.6;
      L     S5T#20M;
      SD    T 6;
      NOP   0;
      NOP   0;
      NOP   0;
      A     T 6;
      =     DB20.DBX 78.0;
NETWORK
TITLE = error discharge time mainscale
      A(;
      ON    M 207.7;
      ON    T 7;
      );
      A     DB10.DBX 57.4;
      AN    M 207.6;
      A     M 2.0;
      L     S5T#3M20S;
      SD    T 7;
      NOP   0;
      NOP   0;
      NOP   0;
      A     T 7;
      =     DB20.DBX 78.2;
NETWORK
TITLE = error discharge time subscale
      A     M 2.0;
      A(;
      ON    M 207.7;
      ON    T 8;
      );
      A     DB11.DBX 57.4;
      AN    M 207.6;
      L     S5T#1M20S;
      SD    T 8;
      NOP   0;
      NOP   0;
      NOP   0;
      A     T 8;
      =     DB20.DBX 78.3;
END_FUNCTION

FUNCTION FC 3 : VOID
TITLE = Dosing, comp. 1
VERSION : 0.1
VAR_TEMP
  dosi_man : BOOL ;
END_VAR
BEGIN
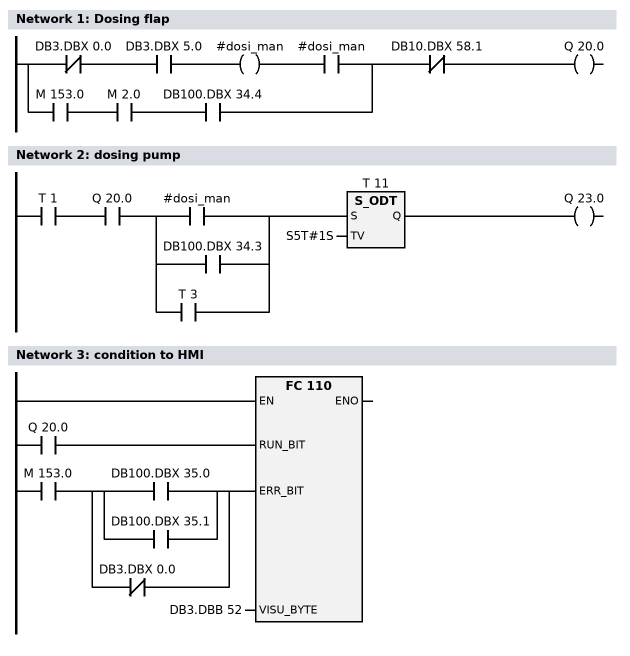
NETWORK
TITLE = Dosing flap
      A(;
      AN    DB3.DBX 0.0;
      A     DB3.DBX 5.0;
      =     #dosi_man;
      A     #dosi_man;
      O;
      A     M 153.0;
      A     M 2.0;
      A     DB100.DBX 34.4;
      );
      AN    DB10.DBX 58.1;
      =     Q 20.0;
NETWORK
TITLE = dosing pump
      A     T 1;
      A     Q 20.0;
      A(;
      O     #dosi_man;
      O     DB100.DBX 34.3;
      O     T 3;
      );
      L     S5T#1S;
      SD    T 11;
      NOP   0;
      NOP   0;
      NOP   0;
      A     T 11;
      =     Q 23.0;
NETWORK
TITLE = condition to HMI 
      A     Q 20.0;
      =     L 1.0;
      BLD   103;
      A     M 153.0;
      A(;
      O     DB100.DBX 35.0;
      O     DB100.DBX 35.1;
      ON    DB3.DBX 0.0;
      );
      =     L 1.1;
      BLD   103;
      CALL  FC 110 (
           RUN_BIT                  := L 1.0,
           ERR_BIT                  := L 1.1,
           VISU_BYTE                := DB3.DBB 52);
      NOP   0;
END_FUNCTION

FUNCTION FC 4 : VOID
TITLE = Dosing, comp. 2
VERSION : 0.1
VAR_TEMP
  dosi_man : BOOL ;
END_VAR
BEGIN
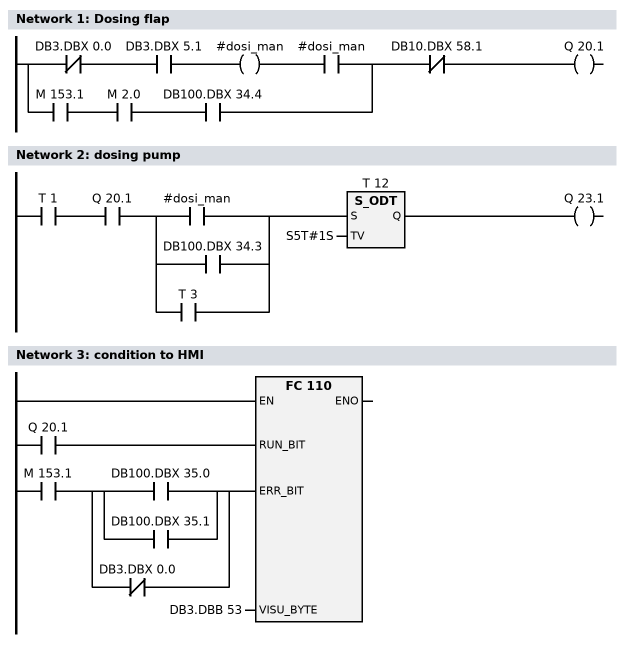
NETWORK
TITLE = Dosing flap
      A(;
      AN    DB3.DBX 0.0;
      A     DB3.DBX 5.1;
      =     #dosi_man;
      A     #dosi_man;
      O;
      A     M 153.1;
      A     M 2.0;
      A     DB100.DBX 34.4;
      );
      AN    DB10.DBX 58.1;
      =     Q 20.1;
NETWORK
TITLE = dosing pump
      A     T 1;
      A     Q 20.1;
      A(;
      O     #dosi_man;
      O     DB100.DBX 34.3;
      O     T 3;
      );
      L     S5T#1S;
      SD    T 12;
      NOP   0;
      NOP   0;
      NOP   0;
      A     T 12;
      =     Q 23.1;
NETWORK
TITLE = condition to HMI 
      A     Q 20.1;
      =     L 1.0;
      BLD   103;
      A     M 153.1;
      A(;
      O     DB100.DBX 35.0;
      O     DB100.DBX 35.1;
      ON    DB3.DBX 0.0;
      );
      =     L 1.1;
      BLD   103;
      CALL  FC 110 (
           RUN_BIT                  := L 1.0,
           ERR_BIT                  := L 1.1,
           VISU_BYTE                := DB3.DBB 53);
      NOP   0;
END_FUNCTION

FUNCTION FC 7 : VOID
TITLE = Dosing component 5
VERSION : 0.1
VAR_TEMP
  dosi_man : BOOL ;
END_VAR
BEGIN
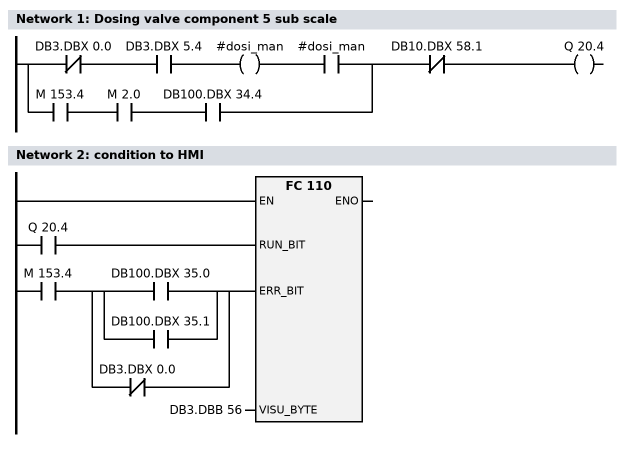
NETWORK
TITLE = Dosing valve component 5 sub scale
//automatic and manual steps
      A(;
      AN    DB3.DBX 0.0;
      A     DB3.DBX 5.4;
      =     #dosi_man;
      A     #dosi_man;
      O;
      A     M 153.4;
      A     M 2.0;
      A     DB100.DBX 34.4;
      );
      AN    DB10.DBX 58.1;
      =     Q 20.4;
NETWORK
TITLE = condition to HMI 
      A     Q 20.4;
      =     L 1.0;
      BLD   103;
      A     M 153.4;
      A(;
      O     DB100.DBX 35.0;
      O     DB100.DBX 35.1;
      ON    DB3.DBX 0.0;
      );
      =     L 1.1;
      BLD   103;
      CALL  FC 110 (
           RUN_BIT                  := L 1.0,
           ERR_BIT                  := L 1.1,
           VISU_BYTE                := DB3.DBB 56);
      NOP   0;
END_FUNCTION

FUNCTION FC 8 : VOID
TITLE = Dosing component 6
VERSION : 0.1
VAR_TEMP
  dosi_man : BOOL ;
END_VAR
BEGIN
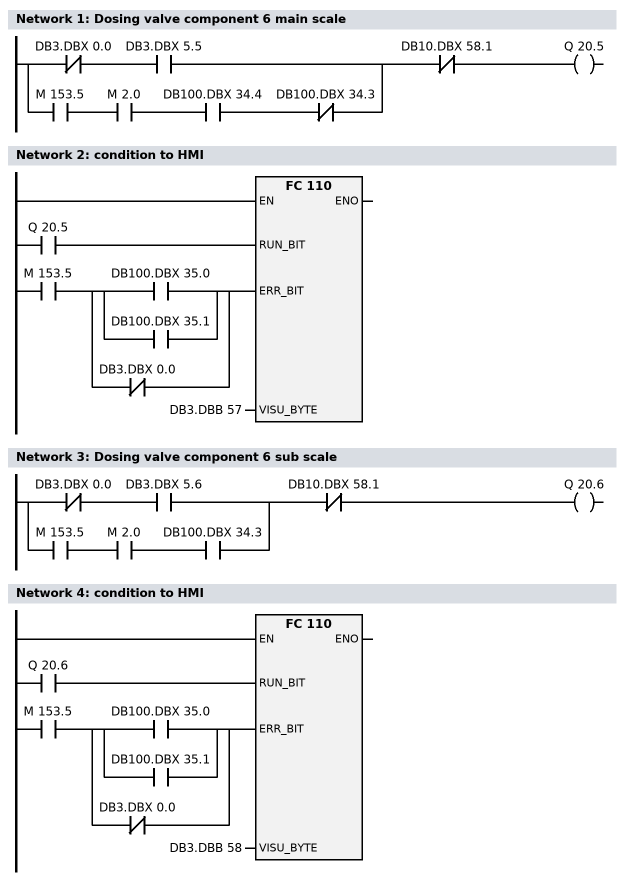
NETWORK
TITLE = Dosing valve component 6 main scale
//automatic and manual steps
      A(;
      AN    DB3.DBX 0.0;
      A     DB3.DBX 5.5;
      O;
      A     M 153.5;
      A     M 2.0;
      A     DB100.DBX 34.4;
      AN    DB100.DBX 34.3;
      );
      AN    DB10.DBX 58.1;
      =     Q 20.5;
NETWORK
TITLE = condition to HMI 
      A     Q 20.5;
      =     L 1.0;
      BLD   103;
      A     M 153.5;
      A(;
      O     DB100.DBX 35.0;
      O     DB100.DBX 35.1;
      ON    DB3.DBX 0.0;
      );
      =     L 1.1;
      BLD   103;
      CALL  FC 110 (
           RUN_BIT                  := L 1.0,
           ERR_BIT                  := L 1.1,
           VISU_BYTE                := DB3.DBB 57);
      NOP   0;
NETWORK
TITLE = Dosing valve component 6 sub scale
//automatic and manual steps
      A(;
      AN    DB3.DBX 0.0;
      A     DB3.DBX 5.6;
      O;
      A     M 153.5;
      A     M 2.0;
      A     DB100.DBX 34.3;
      );
      AN    DB10.DBX 58.1;
      =     Q 20.6;
NETWORK
TITLE = condition to HMI 
      A     Q 20.6;
      =     L 1.0;
      BLD   103;
      A     M 153.5;
      A(;
      O     DB100.DBX 35.0;
      O     DB100.DBX 35.1;
      ON    DB3.DBX 0.0;
      );
      =     L 1.1;
      BLD   103;
      CALL  FC 110 (
           RUN_BIT                  := L 1.0,
           ERR_BIT                  := L 1.1,
           VISU_BYTE                := DB3.DBB 58);
      NOP   0;
END_FUNCTION

FUNCTION FC 9 : VOID
TITLE = Dosing component 7
VERSION : 0.1
VAR_TEMP
  dosi_man : BOOL ;
END_VAR
BEGIN
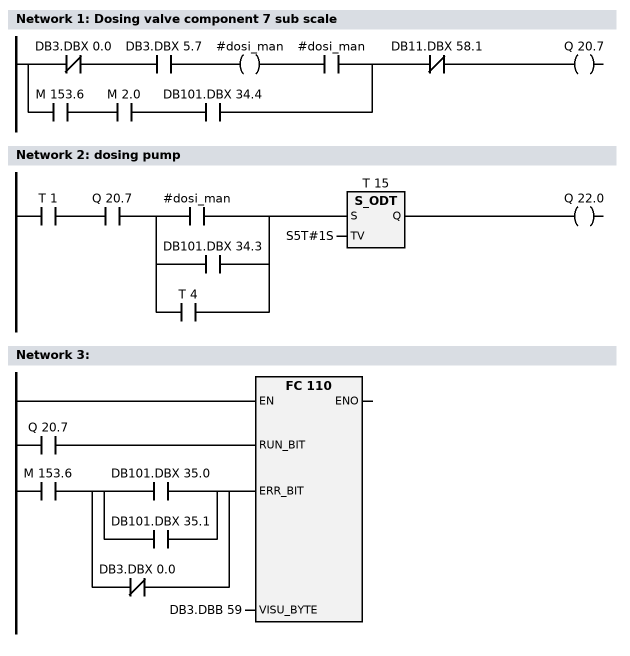
NETWORK
TITLE = Dosing valve component 7 sub scale
//automatic and manual steps
      A(;
      AN    DB3.DBX 0.0;
      A     DB3.DBX 5.7;
      =     #dosi_man;
      A     #dosi_man;
      O;
      A     M 153.6;
      A     M 2.0;
      A     DB101.DBX 34.4;
      );
      AN    DB11.DBX 58.1;
      =     Q 20.7;
NETWORK
TITLE = dosing pump
//automatic and manual steps
      A     T 1;
      A     Q 20.7;
      A(;
      O     #dosi_man;
      O     DB101.DBX 34.3;
      O     T 4;
      );
      L     S5T#1S;
      SD    T 15;
      NOP   0;
      NOP   0;
      NOP   0;
      A     T 15;
      =     Q 22.0;
NETWORK
TITLE =
      A     Q 20.7;
      =     L 1.0;
      BLD   103;
      A     M 153.6;
      A(;
      O     DB101.DBX 35.0;
      O     DB101.DBX 35.1;
      ON    DB3.DBX 0.0;
      );
      =     L 1.1;
      BLD   103;
      CALL  FC 110 (
           RUN_BIT                  := L 1.0,
           ERR_BIT                  := L 1.1,
           VISU_BYTE                := DB3.DBB 59);
      NOP   0;
END_FUNCTION

FUNCTION FC 10 : VOID
TITLE = Dosing component 8
VERSION : 0.1
VAR_TEMP
  dosi_man : BOOL ;
END_VAR
BEGIN
